LIN {X 0,Y 468.927,Z 382.309,A -85,B 0,C 180,E1 -7507.408,E2 -7507.408} C_VEL
LIN {X 0,Y 468.498,Z 392.429,A -85,B 0,C 180,E1 -7508.36,E2 -7508.36} C_VEL
LIN {X 0,Y 467.994,Z 402.327,A -85,B 0,C 180,E1 -7509.516,E2 -7509.516} C_VEL
LIN {X 0,Y 467.657,Z 410.813,A -85,B 0,C 180,E1 -7510.745,E2 -7510.745} C_VEL
LIN {X 0,Y 467.29,Z 417.675,A -85,B 0,C 180,E1 -7511.964,E2 -7511.964} C_VEL
LIN {X 0,Y 467.055,Z 424.349,A -85,B 0,C 180,E1 -7513.461,E2 -7513.461} C_VEL
LIN {X 0,Y 466.861,Z 429.589,A -85,B 0,C 180,E1 -7515.028,E2 -7515.028} C_VEL
LIN {X 0,Y 466.754,Z 432.659,A -85,B 0,C 180,E1 -7516.275,E2 -7516.275} C_VEL
LIN {X 0,Y 466.652,Z 434.866,A -85,B 0,C 180,E1 -7517.551,E2 -7517.551} C_VEL
LIN {X 0,Y 466.622,Z 436.188,A -85,B 0,C 180,E1 -7518.85,E2 -7518.85} C_VEL
LIN {X 0,Y 466.563,Z 436.605,A -85,B 0,C 180,E1 -7520.188,E2 -7520.188} C_VEL
LIN {X 0,Y 466.583,Z 435.757,A -85,B 0,C 180,E1 -7521.861,E2 -7521.861} C_VEL
LIN {X 0,Y 466.695,Z 433.486,A -85,B 0,C 180,E1 -7523.5,E2 -7523.5} C_VEL
LIN {X 0,Y 466.834,Z 429.723,A -85,B 0,C 180,E1 -7525.105,E2 -7525.105} C_VEL
LIN {X 0,Y 467.067,Z 424.472,A -85,B 0,C 180,E1 -7526.687,E2 -7526.687} C_VEL
LIN {X 0,Y 467.35,Z 418.59,A -85,B 0,C 180,E1 -7528.031,E2 -7528.031} C_VEL
LIN {X 0,Y 467.652,Z 411.787,A -85,B 0,C 180,E1 -7529.272,E2 -7529.272} C_VEL
LIN {X 0,Y 468.106,Z 402.57,A -85,B 0,C 180,E1 -7530.624,E2 -7530.624} C_VEL
LIN {X 0,Y 468.57,Z 393.367,A -85,B 0,C 180,E1 -7531.711,E2 -7531.711} C_VEL
LIN {X 0,Y 468.993,Z 383.202,A -85,B 0,C 180,E1 -7532.683,E2 -7532.683} C_VEL
LIN {X 0,Y 469.521,Z 371.519,A -85,B 0,C 180,E1 -7533.572,E2 -7533.572} C_VEL
LIN {X 0,Y 469.906,Z 360.613,A -85,B 0,C 180,E1 -7534.224,E2 -7534.224} C_VEL
LIN {X 0,Y 470.276,Z 347.828,A -85,B 0,C 180,E1 -7534.792,E2 -7534.792} C_VEL
LIN {X 0,Y 470.547,Z 334.524,A -85,B 0,C 180,E1 -7535.191,E2 -7535.191} C_VEL
LIN {X 0,Y 471.448,Z 240.188,A -85,B 0,C 180,E1 -7536.74,E2 -7536.74} C_VEL
LIN {X 0,Y 468.543,Z 226.096,A -85,B 0,C 180,E1 -7537.105,E2 -7537.105} C_VEL
LIN {X 0,Y 468.569,Z 216.391,A -85,B 0,C 180,E1 -7538.902,E2 -7538.902} C_VEL
LIN {X 0,Y 467.611,Z 211.239,A -85,B 0,C 180,E1 -7539.949,E2 -7539.949} C_VEL
LIN {X 0,Y 467.572,Z 211.241,A -85,B 0,C 180,E1 -7542.506,E2 -7542.506} C_VEL
LIN {X 0,Y 467.561,Z 211.248,A -85,B 0,C 180,E1 -7545.195,E2 -7545.195} C_VEL
LIN {X 0,Y 467.648,Z 211.236,A -85,B 0,C 180,E1 -7547.855,E2 -7547.855} C_VEL
LIN {X 0,Y 467.633,Z 211.238,A -85,B 0,C 180,E1 -7551.357,E2 -7551.357} C_VEL
LIN {X 0,Y 467.71,Z 211.223,A -85,B 0,C 180,E1 -7553.962,E2 -7553.962} C_VEL
LIN {X 0,Y 467.808,Z 211.214,A -85,B 0,C 180,E1 -7557.417,E2 -7557.417} C_VEL
LIN {X 0,Y 467.826,Z 211.208,A -85,B 0,C 180,E1 -7560,E2 -7560} C_VEL
LIN {X 0,Y 467.806,Z 211.213,A -85,B 0,C 180,E1 -7562.583,E2 -7562.583} C_VEL
LIN {X 0,Y 467.681,Z 211.223,A -85,B 0,C 180,E1 -7566.038,E2 -7566.038} C_VEL
LIN {X 0,Y 467.632,Z 211.235,A -85,B 0,C 180,E1 -7568.644,E2 -7568.644} C_VEL
LIN {X 0,Y 467.634,Z 211.23,A -85,B 0,C 180,E1 -7572.146,E2 -7572.146} C_VEL
LIN {X 0,Y 467.619,Z 211.233,A -85,B 0,C 180,E1 -7575.894,E2 -7575.894} C_VEL
LIN {X 0,Y 467.578,Z 211.238,A -85,B 0,C 180,E1 -7579.31,E2 -7579.31} C_VEL
LIN {X 0,Y 467.497,Z 211.25,A -85,B 0,C 180,E1 -7582.076,E2 -7582.076} C_VEL
LIN {X 0,Y 467.563,Z 211.244,A -85,B 0,C 180,E1 -7584.89,E2 -7584.89} C_VEL
LIN {X 0,Y 467.58,Z 211.237,A -85,B 0,C 180,E1 -7587.772,E2 -7587.772} C_VEL
LIN {X 0,Y 467.53,Z 211.245,A -85,B 0,C 180,E1 -7591.048,E2 -7591.048} C_VEL
LIN {X 0,Y 467.555,Z 211.246,A -85,B 0,C 180,E1 -7594.245,E2 -7594.245} C_VEL
LIN {X 0,Y 467.517,Z 211.246,A -85,B 0,C 180,E1 -7597.189,E2 -7597.189} C_VEL
LIN {X 0,Y 467.545,Z 211.247,A -85,B 0,C 180,E1 -7600.268,E2 -7600.268} C_VEL
LIN {X 0,Y 467.561,Z 211.242,A -85,B 0,C 180,E1 -7602.57,E2 -7602.57} C_VEL
LIN {X 0,Y 467.541,Z 211.242,A -85,B 0,C 180,E1 -7605.056,E2 -7605.056} C_VEL
LIN {X 0,Y 467.568,Z 211.24,A -85,B 0,C 180,E1 -7607.443,E2 -7607.443} C_VEL
LIN {X 0,Y 467.563,Z 211.241,A -85,B 0,C 180,E1 -7610.858,E2 -7610.858} C_VEL
LIN {X 0,Y 467.547,Z 211.247,A -85,B 0,C 180,E1 -7614.264,E2 -7614.264} C_VEL
LIN {X 0,Y 467.569,Z 211.242,A -85,B 0,C 180,E1 -7617.324,E2 -7617.324} C_VEL
LIN {X 0,Y 467.559,Z 211.245,A -85,B 0,C 180,E1 -7620.671,E2 -7620.671} C_VEL
LIN {X 0,Y 467.649,Z 211.353,A -85,B 0,C 180,E1 -7623.806,E2 -7623.806} C_VEL
LIN {X 0,Y 469.751,Z 222.852,A -85,B 0,C 180,E1 -7625.872,E2 -7625.872} C_VEL
LIN {X 0,Y 469.241,Z 237.693,A -85,B 0,C 180,E1 -7628.337,E2 -7628.337} C_VEL
LIN {X 0,Y 468.466,Z 259.202,A -85,B 0,C 180,E1 -7631.865,E2 -7631.865} C_VEL
LIN {X 0,Y 468.239,Z 265.745,A -85,B 0,C 180,E1 -7632.93,E2 -7632.93} C_VEL
LIN {X 0,Y 471.203,Z 287.173,A -85,B 0,C 180,E1 -7633.401,E2 -7633.401} C_VEL
LIN {X 0,Y 470.387,Z 375.627,A -85,B 0,C 180,E1 -7634.845,E2 -7634.845} C_VEL
LIN {X 0,Y 470.003,Z 387.734,A -85,B 0,C 180,E1 -7635.192,E2 -7635.192} C_VEL
LIN {X 0,Y 469.51,Z 401.066,A -85,B 0,C 180,E1 -7635.758,E2 -7635.758} C_VEL
LIN {X 0,Y 469.007,Z 413.098,A -85,B 0,C 180,E1 -7636.461,E2 -7636.461} C_VEL
LIN {X 0,Y 468.591,Z 424.153,A -85,B 0,C 180,E1 -7637.289,E2 -7637.289} C_VEL
LIN {X 0,Y 468.088,Z 435.073,A -85,B 0,C 180,E1 -7638.307,E2 -7638.307} C_VEL
LIN {X 0,Y 467.598,Z 444.443,A -85,B 0,C 180,E1 -7639.391,E2 -7639.391} C_VEL
LIN {X 0,Y 467.237,Z 453.554,A -85,B 0,C 180,E1 -7640.696,E2 -7640.696} C_VEL
LIN {X 0,Y 466.979,Z 460.9,A -85,B 0,C 180,E1 -7641.999,E2 -7641.999} C_VEL
LIN {X 0,Y 466.828,Z 465.861,A -85,B 0,C 180,E1 -7643.083,E2 -7643.083} C_VEL
LIN {X 0,Y 466.727,Z 470.686,A -85,B 0,C 180,E1 -7644.384,E2 -7644.384} C_VEL
LIN {X 0,Y 466.657,Z 474.379,A -85,B 0,C 180,E1 -7645.682,E2 -7645.682} C_VEL
LIN {X 0,Y 466.697,Z 476.289,A -85,B 0,C 180,E1 -7646.547,E2 -7646.547} C_VEL
LIN {X 0,Y 466.681,Z 477.722,A -85,B 0,C 180,E1 -7647.411,E2 -7647.411} C_VEL
LIN {X 0,Y 466.661,Z 478.748,A -85,B 0,C 180,E1 -7648.274,E2 -7648.274} C_VEL
LIN {X 0,Y 466.624,Z 479.377,A -85,B 0,C 180,E1 -7649.137,E2 -7649.137} C_VEL
LIN {X 0,Y 466.607,Z 479.604,A -85,B 0,C 180,E1 -7650,E2 -7650} C_VEL
LIN {X 0,Y 466.624,Z 479.391,A -85,B 0,C 180,E1 -7650.863,E2 -7650.863} C_VEL
LIN {X 0,Y 466.661,Z 478.783,A -85,B 0,C 180,E1 -7651.726,E2 -7651.726} C_VEL
LIN {X 0,Y 466.68,Z 477.779,A -85,B 0,C 180,E1 -7652.589,E2 -7652.589} C_VEL
LIN {X 0,Y 466.691,Z 476.357,A -85,B 0,C 180,E1 -7653.453,E2 -7653.453} C_VEL
LIN {X 0,Y 466.688,Z 473.375,A -85,B 0,C 180,E1 -7654.75,E2 -7654.75} C_VEL
LIN {X 0,Y 466.743,Z 469.333,A -85,B 0,C 180,E1 -7656.05,E2 -7656.05} C_VEL
LIN {X 0,Y 466.906,Z 463.103,A -85,B 0,C 180,E1 -7657.567,E2 -7657.567} C_VEL
LIN {X 0,Y 467.132,Z 456.305,A -85,B 0,C 180,E1 -7658.87,E2 -7658.87} C_VEL
LIN {X 0,Y 467.435,Z 447.857,A -85,B 0,C 180,E1 -7660.174,E2 -7660.174} C_VEL
LIN {X 0,Y 467.869,Z 439.152,A -85,B 0,C 180,E1 -7661.26,E2 -7661.26} C_VEL
LIN {X 0,Y 468.308,Z 428.98,A -85,B 0,C 180,E1 -7662.295,E2 -7662.295} C_VEL
LIN {X 0,Y 468.853,Z 417.789,A -85,B 0,C 180,E1 -7663.213,E2 -7663.213} C_VEL
LIN {X 0,Y 469.3,Z 405.934,A -85,B 0,C 180,E1 -7663.972,E2 -7663.972} C_VEL
LIN {X 0,Y 469.775,Z 393.641,A -85,B 0,C 180,E1 -7664.566,E2 -7664.566} C_VEL
LIN {X 0,Y 470.19,Z 380.174,A -85,B 0,C 180,E1 -7665.023,E2 -7665.023} C_VEL
LIN {X 0,Y 470.485,Z 365.01,A -85,B 0,C 180,E1 -7665.318,E2 -7665.318} C_VEL
LIN {X 0,Y 471.003,Z 285.344,A -85,B 0,C 180,E1 -7666.59,E2 -7666.59} C_VEL
LIN {X 0,Y 468.3,Z 266.657,A -85,B 0,C 180,E1 -7667.015,E2 -7667.015} C_VEL
LIN {X 0,Y 468.98,Z 247.902,A -85,B 0,C 180,E1 -7670.159,E2 -7670.159} C_VEL
LIN {X 0,Y 469.761,Z 230.47,A -85,B 0,C 180,E1 -7673.121,E2 -7673.121} C_VEL
LIN {X 0,Y 470.065,Z 224.101,A -85,B 0,C 180,E1 -7674.213,E2 -7674.213} C_VEL
LIN {X 0,Y 467.962,Z 212.85,A -85,B 0,C 180,E1 -7676.294,E2 -7676.294} C_VEL
LIN {X 0,Y 467.646,Z 211.235,A -85,B 0,C 180,E1 -7676.614,E2 -7676.614} C_VEL
LIN {X 0,Y 467.542,Z 211.247,A -85,B 0,C 180,E1 -7679.735,E2 -7679.735} C_VEL
LIN {X 0,Y 467.57,Z 211.238,A -85,B 0,C 180,E1 -7682.755,E2 -7682.755} C_VEL
LIN {X 0,Y 467.539,Z 211.249,A -85,B 0,C 180,E1 -7685.886,E2 -7685.886} C_VEL
LIN {X 0,Y 467.562,Z 211.239,A -85,B 0,C 180,E1 -7689.141,E2 -7689.141} C_VEL
LIN {X 0,Y 467.564,Z 211.239,A -85,B 0,C 180,E1 -7692.564,E2 -7692.564} C_VEL
LIN {X 0,Y 467.544,Z 211.242,A -85,B 0,C 180,E1 -7695.049,E2 -7695.049} C_VEL
LIN {X 0,Y 467.562,Z 211.243,A -85,B 0,C 180,E1 -7697.436,E2 -7697.436} C_VEL
LIN {X 0,Y 467.528,Z 211.243,A -85,B 0,C 180,E1 -7700.85,E2 -7700.85} C_VEL
LIN {X 0,Y 467.529,Z 211.244,A -85,B 0,C 180,E1 -7704.257,E2 -7704.257} C_VEL
LIN {X 0,Y 467.546,Z 211.246,A -85,B 0,C 180,E1 -7707.318,E2 -7707.318} C_VEL
LIN {X 0,Y 467.529,Z 211.243,A -85,B 0,C 180,E1 -7710.665,E2 -7710.665} C_VEL
LIN {X 0,Y 467.575,Z 211.242,A -85,B 0,C 180,E1 -7713.197,E2 -7713.197} C_VEL
LIN {X 0,Y 467.55,Z 211.24,A -85,B 0,C 180,E1 -7716.466,E2 -7716.466} C_VEL
LIN {X 0,Y 467.576,Z 211.24,A -85,B 0,C 180,E1 -7719.775,E2 -7719.775} C_VEL
LIN {X 0,Y 467.564,Z 211.239,A -85,B 0,C 180,E1 -7722.505,E2 -7722.505} C_VEL
LIN {X 0,Y 467.555,Z 211.248,A -85,B 0,C 180,E1 -7725.194,E2 -7725.194} C_VEL
LIN {X 0,Y 467.632,Z 211.231,A -85,B 0,C 180,E1 -7727.854,E2 -7727.854} C_VEL
LIN {X 0,Y 467.631,Z 211.235,A -85,B 0,C 180,E1 -7731.356,E2 -7731.356} C_VEL
LIN {X 0,Y 467.681,Z 211.224,A -85,B 0,C 180,E1 -7733.961,E2 -7733.961} C_VEL
LIN {X 0,Y 467.805,Z 211.211,A -85,B 0,C 180,E1 -7737.416,E2 -7737.416} C_VEL
LIN {X 0,Y 467.825,Z 211.206,A -85,B 0,C 180,E1 -7740,E2 -7740} C_VEL
LIN {X 0,Y 467.807,Z 211.213,A -85,B 0,C 180,E1 -7742.583,E2 -7742.583} C_VEL
LIN {X 0,Y 467.709,Z 211.221,A -85,B 0,C 180,E1 -7746.038,E2 -7746.038} C_VEL
LIN {X 0,Y 467.632,Z 211.237,A -85,B 0,C 180,E1 -7748.643,E2 -7748.643} C_VEL
LIN {X 0,Y 467.647,Z 211.23,A -85,B 0,C 180,E1 -7752.145,E2 -7752.145} C_VEL
LIN {X 0,Y 467.617,Z 211.233,A -85,B 0,C 180,E1 -7755.894,E2 -7755.894} C_VEL
LIN {X 0,Y 467.581,Z 211.237,A -85,B 0,C 180,E1 -7759.309,E2 -7759.309} C_VEL
LIN {X 0,Y 467.575,Z 211.24,A -85,B 0,C 180,E1 -7762.071,E2 -7762.071} C_VEL
LIN {X 0,Y 467.572,Z 211.24,A -85,B 0,C 180,E1 -7764.889,E2 -7764.889} C_VEL
LIN {X 0,Y 467.586,Z 211.237,A -85,B 0,C 180,E1 -7767.771,E2 -7767.771} C_VEL
LIN {X 0,Y 467.531,Z 211.243,A -85,B 0,C 180,E1 -7771.048,E2 -7771.048} C_VEL
LIN {X 0,Y 467.552,Z 211.248,A -85,B 0,C 180,E1 -7774.245,E2 -7774.245} C_VEL
LIN {X 0,Y 467.515,Z 211.245,A -85,B 0,C 180,E1 -7777.19,E2 -7777.19} C_VEL
LIN {X 0,Y 467.57,Z 211.245,A -85,B 0,C 180,E1 -7780.265,E2 -7780.265} C_VEL
LIN {X 0,Y 467.589,Z 211.238,A -85,B 0,C 180,E1 -7782.574,E2 -7782.574} C_VEL
LIN {X 0,Y 467.541,Z 211.241,A -85,B 0,C 180,E1 -7785.056,E2 -7785.056} C_VEL
LIN {X 0,Y 467.563,Z 211.24,A -85,B 0,C 180,E1 -7787.443,E2 -7787.443} C_VEL
LIN {X 0,Y 467.577,Z 211.237,A -85,B 0,C 180,E1 -7790.86,E2 -7790.86} C_VEL
LIN {X 0,Y 467.543,Z 211.245,A -85,B 0,C 180,E1 -7794.263,E2 -7794.263} C_VEL
LIN {X 0,Y 467.565,Z 211.24,A -85,B 0,C 180,E1 -7797.324,E2 -7797.324} C_VEL
LIN {X 0,Y 467.562,Z 211.239,A -85,B 0,C 180,E1 -7800.669,E2 -7800.669} C_VEL
LIN {X 0,Y 467.615,Z 211.234,A -85,B 0,C 180,E1 -7803.203,E2 -7803.203} C_VEL
LIN {X 0,Y 467.583,Z 211.236,A -85,B 0,C 180,E1 -7806.47,E2 -7806.47} C_VEL
LIN {X 0,Y 467.614,Z 211.238,A -85,B 0,C 180,E1 -7809.779,E2 -7809.779} C_VEL
LIN {X 0,Y 467.602,Z 211.234,A -85,B 0,C 180,E1 -7812.509,E2 -7812.509} C_VEL
LIN {X 0,Y 467.604,Z 211.238,A -85,B 0,C 180,E1 -7815.198,E2 -7815.198} C_VEL
LIN {X 0,Y 467.594,Z 211.237,A -85,B 0,C 180,E1 -7815.47,E2 -7815.47} C_VEL
LIN {X 0,Y 466.926,Z 211.32,A -85,B 0,C 180,E1 -7816.189,E2 -7816.189} C_VEL
LIN {X 0,Y 464.08,Z 211.68,A -85,B 0,C 180,E1 -7817.357,E2 -7817.357} C_VEL
LIN {X 0,Y 461.679,Z 211.974,A -85,B 0,C 180,E1 -7818.299,E2 -7818.299} C_VEL
LIN {X 0,Y 460.654,Z 212.102,A -85,B 0,C 180,E1 -7819.027,E2 -7819.027} C_VEL
LIN {X 0,Y 460.574,Z 212.114,A -85,B 0,C 180,E1 -7819.273,E2 -7819.273} C_VEL
LIN {X 0,Y 460.713,Z 212.092,A -85,B 0,C 180,E1 -7822.544,E2 -7822.544} C_VEL
LIN {X 0,Y 460.693,Z 212.096,A -85,B 0,C 180,E1 -7824.749,E2 -7824.749} C_VEL
LIN {X 0,Y 460.823,Z 212.085,A -85,B 0,C 180,E1 -7827.378,E2 -7827.378} C_VEL
LIN {X 0,Y 460.851,Z 212.075,A -85,B 0,C 180,E1 -7830,E2 -7830} C_VEL
LIN {X 0,Y 460.823,Z 212.08,A -85,B 0,C 180,E1 -7832.622,E2 -7832.622} C_VEL
LIN {X 0,Y 460.692,Z 212.095,A -85,B 0,C 180,E1 -7836.13,E2 -7836.13} C_VEL
LIN {X 0,Y 460.626,Z 212.107,A -85,B 0,C 180,E1 -7838.775,E2 -7838.775} C_VEL
LIN {X 0,Y 460.61,Z 212.107,A -85,B 0,C 180,E1 -7842.444,E2 -7842.444} C_VEL
LIN {X 0,Y 460.595,Z 212.107,A -85,B 0,C 180,E1 -7845.996,E2 -7845.996} C_VEL
LIN {X 0,Y 460.565,Z 212.118,A -85,B 0,C 180,E1 -7848.9,E2 -7848.9} C_VEL
LIN {X 0,Y 460.508,Z 212.118,A -85,B 0,C 180,E1 -7851.484,E2 -7851.484} C_VEL
LIN {X 0,Y 460.533,Z 212.117,A -85,B 0,C 180,E1 -7854.33,E2 -7854.33} C_VEL
LIN {X 0,Y 460.572,Z 212.114,A -85,B 0,C 180,E1 -7857.241,E2 -7857.241} C_VEL
LIN {X 0,Y 460.625,Z 212.228,A -85,B 0,C 180,E1 -7859.808,E2 -7859.808} C_VEL
LIN {X 0,Y 461.644,Z 218.347,A -85,B 0,C 180,E1 -7861.168,E2 -7861.168} C_VEL
LIN {X 0,Y 461.512,Z 226.254,A -85,B 0,C 180,E1 -7862.829,E2 -7862.829} C_VEL
LIN {X 0,Y 464.399,Z 240.609,A -85,B 0,C 180,E1 -7863.185,E2 -7863.185} C_VEL
LIN {X 0,Y 463.53,Z 333.526,A -85,B 0,C 180,E1 -7864.712,E2 -7864.712} C_VEL
LIN {X 0,Y 463.213,Z 346.696,A -85,B 0,C 180,E1 -7865.101,E2 -7865.101} C_VEL
LIN {X 0,Y 462.969,Z 358.713,A -85,B 0,C 180,E1 -7865.625,E2 -7865.625} C_VEL
LIN {X 0,Y 462.513,Z 370.891,A -85,B 0,C 180,E1 -7866.338,E2 -7866.338} C_VEL
LIN {X 0,Y 461.998,Z 382.253,A -85,B 0,C 180,E1 -7867.201,E2 -7867.201} C_VEL
LIN {X 0,Y 461.495,Z 393.331,A -85,B 0,C 180,E1 -7868.259,E2 -7868.259} C_VEL
LIN {X 0,Y 460.996,Z 402.697,A -85,B 0,C 180,E1 -7869.377,E2 -7869.377} C_VEL
LIN {X 0,Y 460.658,Z 411.115,A -85,B 0,C 180,E1 -7870.615,E2 -7870.615} C_VEL
LIN {X 0,Y 460.251,Z 418.028,A -85,B 0,C 180,E1 -7871.861,E2 -7871.861} C_VEL
LIN {X 0,Y 460.052,Z 423.596,A -85,B 0,C 180,E1 -7873.102,E2 -7873.102} C_VEL
LIN {X 0,Y 459.825,Z 429.07,A -85,B 0,C 180,E1 -7874.667,E2 -7874.667} C_VEL
LIN {X 0,Y 459.711,Z 432.36,A -85,B 0,C 180,E1 -7875.927,E2 -7875.927} C_VEL
LIN {X 0,Y 459.55,Z 435.433,A -85,B 0,C 180,E1 -7877.709,E2 -7877.709} C_VEL
LIN {X 0,Y 459.527,Z 436.537,A -85,B 0,C 180,E1 -7878.88,E2 -7878.88} C_VEL
LIN {X 0,Y 459.489,Z 436.946,A -85,B 0,C 180,E1 -7880.029,E2 -7880.029} C_VEL
LIN {X 0,Y 459.478,Z 436.581,A -85,B 0,C 180,E1 -7881.26,E2 -7881.26} C_VEL
LIN {X 0,Y 459.514,Z 435.203,A -85,B 0,C 180,E1 -7882.676,E2 -7882.676} C_VEL
LIN {X 0,Y 459.678,Z 432.697,A -85,B 0,C 180,E1 -7884.118,E2 -7884.118} C_VEL
LIN {X 0,Y 459.807,Z 428.84,A -85,B 0,C 180,E1 -7885.617,E2 -7885.617} C_VEL
LIN {X 0,Y 460.092,Z 423.407,A -85,B 0,C 180,E1 -7887.145,E2 -7887.145} C_VEL
LIN {X 0,Y 460.399,Z 417.313,A -85,B 0,C 180,E1 -7888.479,E2 -7888.479} C_VEL
LIN {X 0,Y 460.784,Z 409.913,A -85,B 0,C 180,E1 -7889.78,E2 -7889.78} C_VEL
LIN {X 0,Y 461.267,Z 400.737,A -85,B 0,C 180,E1 -7891.07,E2 -7891.07} C_VEL
LIN {X 0,Y 461.727,Z 390.638,A -85,B 0,C 180,E1 -7892.213,E2 -7892.213} C_VEL
LIN {X 0,Y 462.284,Z 379.757,A -85,B 0,C 180,E1 -7893.198,E2 -7893.198} C_VEL
LIN {X 0,Y 462.807,Z 367.681,A -85,B 0,C 180,E1 -7894.054,E2 -7894.054} C_VEL
LIN {X 0,Y 463.221,Z 356.195,A -85,B 0,C 180,E1 -7894.681,E2 -7894.681} C_VEL
LIN {X 0,Y 463.538,Z 343.535,A -85,B 0,C 180,E1 -7895.186,E2 -7895.186} C_VEL
LIN {X 0,Y 463.781,Z 329.939,A -85,B 0,C 180,E1 -7895.529,E2 -7895.529} C_VEL
LIN {X 0,Y 464.699,Z 241.15,A -85,B 0,C 180,E1 -7896.993,E2 -7896.993} C_VEL
LIN {X 0,Y 461.648,Z 226.372,A -85,B 0,C 180,E1 -7897.394,E2 -7897.394} C_VEL
LIN {X 0,Y 461.632,Z 217.605,A -85,B 0,C 180,E1 -7899.037,E2 -7899.037} C_VEL
LIN {X 0,Y 460.568,Z 212.116,A -85,B 0,C 180,E1 -7900.153,E2 -7900.153} C_VEL
LIN {X 0,Y 460.527,Z 212.123,A -85,B 0,C 180,E1 -7903.145,E2 -7903.145} C_VEL
LIN {X 0,Y 460.515,Z 212.125,A -85,B 0,C 180,E1 -7905.867,E2 -7905.867} C_VEL
LIN {X 0,Y 460.589,Z 212.114,A -85,B 0,C 180,E1 -7908.559,E2 -7908.559} C_VEL
LIN {X 0,Y 460.647,Z 212.103,A -85,B 0,C 180,E1 -7912.108,E2 -7912.108} C_VEL
LIN {X 0,Y 460.656,Z 212.104,A -85,B 0,C 180,E1 -7914.748,E2 -7914.748} C_VEL
LIN {X 0,Y 460.749,Z 212.094,A -85,B 0,C 180,E1 -7917.378,E2 -7917.378} C_VEL
LIN {X 0,Y 460.797,Z 212.084,A -85,B 0,C 180,E1 -7920,E2 -7920} C_VEL
LIN {X 0,Y 460.748,Z 212.093,A -85,B 0,C 180,E1 -7922.623,E2 -7922.623} C_VEL
LIN {X 0,Y 460.648,Z 212.099,A -85,B 0,C 180,E1 -7926.131,E2 -7926.131} C_VEL
LIN {X 0,Y 460.58,Z 212.113,A -85,B 0,C 180,E1 -7928.777,E2 -7928.777} C_VEL
LIN {X 0,Y 460.588,Z 212.11,A -85,B 0,C 180,E1 -7932.458,E2 -7932.458} C_VEL
LIN {X 0,Y 460.577,Z 212.11,A -85,B 0,C 180,E1 -7936.009,E2 -7936.009} C_VEL
LIN {X 0,Y 460.524,Z 212.116,A -85,B 0,C 180,E1 -7939.618,E2 -7939.618} C_VEL
LIN {X 0,Y 460.472,Z 212.129,A -85,B 0,C 180,E1 -7942.431,E2 -7942.431} C_VEL
LIN {X 0,Y 460.527,Z 212.117,A -85,B 0,C 180,E1 -7945.804,E2 -7945.804} C_VEL
LIN {X 0,Y 460.513,Z 212.121,A -85,B 0,C 180,E1 -7948.236,E2 -7948.236} C_VEL
LIN {X 0,Y 460.484,Z 212.122,A -85,B 0,C 180,E1 -7951.286,E2 -7951.286} C_VEL
LIN {X 0,Y 460.5,Z 212.124,A -85,B 0,C 180,E1 -7954.509,E2 -7954.509} C_VEL
LIN {X 0,Y 460.47,Z 212.124,A -85,B 0,C 180,E1 -7957.626,E2 -7957.626} C_VEL
LIN {X 0,Y 460.51,Z 212.123,A -85,B 0,C 180,E1 -7960.272,E2 -7960.272} C_VEL
LIN {X 0,Y 460.47,Z 212.122,A -85,B 0,C 180,E1 -7963.379,E2 -7963.379} C_VEL
LIN {X 0,Y 460.473,Z 212.125,A -85,B 0,C 180,E1 -7966.627,E2 -7966.627} C_VEL
LIN {X 0,Y 460.522,Z 212.12,A -85,B 0,C 180,E1 -7969.734,E2 -7969.734} C_VEL
LIN {X 0,Y 460.483,Z 212.125,A -85,B 0,C 180,E1 -7972.527,E2 -7972.527} C_VEL
LIN {X 0,Y 460.534,Z 212.119,A -85,B 0,C 180,E1 -7975.627,E2 -7975.627} C_VEL
LIN {X 0,Y 460.526,Z 212.119,A -85,B 0,C 180,E1 -7978.747,E2 -7978.747} C_VEL
LIN {X 0,Y 460.572,Z 212.118,A -85,B 0,C 180,E1 -7982.257,E2 -7982.257} C_VEL
LIN {X 0,Y 460.601,Z 212.258,A -85,B 0,C 180,E1 -7983.588,E2 -7983.588} C_VEL
LIN {X 0,Y 462.485,Z 221.848,A -85,B 0,C 180,E1 -7985.349,E2 -7985.349} C_VEL
LIN {X 0,Y 462.843,Z 225.754,A -85,B 0,C 180,E1 -7986.037,E2 -7986.037} C_VEL
LIN {X 0,Y 462.101,Z 242.367,A -85,B 0,C 180,E1 -7988.828,E2 -7988.828} C_VEL
LIN {X 0,Y 461.371,Z 263.03,A -85,B 0,C 180,E1 -7992.264,E2 -7992.264} C_VEL
LIN {X 0,Y 461.288,Z 265.345,A -85,B 0,C 180,E1 -7992.646,E2 -7992.646} C_VEL
LIN {X 0,Y 464.425,Z 287.456,A -85,B 0,C 180,E1 -7993.15,E2 -7993.15} C_VEL
LIN {X 0,Y 463.543,Z 375.457,A -85,B 0,C 180,E1 -7994.615,E2 -7994.615} C_VEL
LIN {X 0,Y 463.121,Z 388.241,A -85,B 0,C 180,E1 -7994.995,E2 -7994.995} C_VEL
LIN {X 0,Y 462.599,Z 400.776,A -85,B 0,C 180,E1 -7995.54,E2 -7995.54} C_VEL
LIN {X 0,Y 462.085,Z 412.792,A -85,B 0,C 180,E1 -7996.254,E2 -7996.254} C_VEL
LIN {X 0,Y 461.589,Z 424.834,A -85,B 0,C 180,E1 -7997.178,E2 -7997.178} C_VEL
LIN {X 0,Y 461.1,Z 434.754,A -85,B 0,C 180,E1 -7998.127,E2 -7998.127} C_VEL
LIN {X 0,Y 460.586,Z 444.117,A -85,B 0,C 180,E1 -7999.228,E2 -7999.228} C_VEL
LIN {X 0,Y 460.177,Z 453.224,A -85,B 0,C 180,E1 -8000.552,E2 -8000.552} C_VEL
LIN {X 0,Y 459.906,Z 460.57,A -85,B 0,C 180,E1 -8001.875,E2 -8001.875} C_VEL
LIN {X 0,Y 459.72,Z 466.815,A -85,B 0,C 180,E1 -8003.295,E2 -8003.295} C_VEL
LIN {X 0,Y 459.64,Z 471.707,A -85,B 0,C 180,E1 -8004.737,E2 -8004.737} C_VEL
LIN {X 0,Y 459.572,Z 474.055,A -85,B 0,C 180,E1 -8005.615,E2 -8005.615} C_VEL
LIN {X 0,Y 459.594,Z 475.965,A -85,B 0,C 180,E1 -8006.494,E2 -8006.494} C_VEL
LIN {X 0,Y 459.601,Z 477.398,A -85,B 0,C 180,E1 -8007.371,E2 -8007.371} C_VEL
LIN {X 0,Y 459.57,Z 478.423,A -85,B 0,C 180,E1 -8008.247,E2 -8008.247} C_VEL
LIN {X 0,Y 459.557,Z 479.053,A -85,B 0,C 180,E1 -8009.124,E2 -8009.124} C_VEL
LIN {X 0,Y 459.538,Z 479.277,A -85,B 0,C 180,E1 -8010,E2 -8010} C_VEL
LIN {X 0,Y 459.557,Z 479.061,A -85,B 0,C 180,E1 -8010.876,E2 -8010.876} C_VEL
LIN {X 0,Y 459.57,Z 478.45,A -85,B 0,C 180,E1 -8011.752,E2 -8011.752} C_VEL
LIN {X 0,Y 459.6,Z 477.443,A -85,B 0,C 180,E1 -8012.629,E2 -8012.629} C_VEL
LIN {X 0,Y 459.589,Z 476.013,A -85,B 0,C 180,E1 -8013.506,E2 -8013.506} C_VEL
LIN {X 0,Y 459.618,Z 473.025,A -85,B 0,C 180,E1 -8014.824,E2 -8014.824} C_VEL
LIN {X 0,Y 459.714,Z 467.911,A -85,B 0,C 180,E1 -8016.43,E2 -8016.43} C_VEL
LIN {X 0,Y 459.87,Z 461.699,A -85,B 0,C 180,E1 -8017.905,E2 -8017.905} C_VEL
LIN {X 0,Y 460.152,Z 454.642,A -85,B 0,C 180,E1 -8019.227,E2 -8019.227} C_VEL
LIN {X 0,Y 460.491,Z 445.789,A -85,B 0,C 180,E1 -8020.552,E2 -8020.552} C_VEL
LIN {X 0,Y 461.058,Z 435.745,A -85,B 0,C 180,E1 -8021.762,E2 -8021.762} C_VEL
LIN {X 0,Y 461.561,Z 424.877,A -85,B 0,C 180,E1 -8022.806,E2 -8022.806} C_VEL
LIN {X 0,Y 462.04,Z 414.123,A -85,B 0,C 180,E1 -8023.635,E2 -8023.635} C_VEL
LIN {X 0,Y 462.553,Z 402.351,A -85,B 0,C 180,E1 -8024.349,E2 -8024.349} C_VEL
LIN {X 0,Y 463.027,Z 389.502,A -85,B 0,C 180,E1 -8024.923,E2 -8024.923} C_VEL
LIN {X 0,Y 463.403,Z 375.882,A -85,B 0,C 180,E1 -8025.333,E2 -8025.333} C_VEL
LIN {X 0,Y 464.134,Z 301.407,A -85,B 0,C 180,E1 -8026.559,E2 -8026.559} C_VEL
LIN {X 0,Y 464.135,Z 286.017,A -85,B 0,C 180,E1 -8026.816,E2 -8026.816} C_VEL
LIN {X 0,Y 461.311,Z 266.427,A -85,B 0,C 180,E1 -8027.256,E2 -8027.256} C_VEL
LIN {X 0,Y 462.007,Z 248.892,A -85,B 0,C 180,E1 -8030.245,E2 -8030.245} C_VEL
LIN {X 0,Y 462.824,Z 231.449,A -85,B 0,C 180,E1 -8033.251,E2 -8033.251} C_VEL
LIN {X 0,Y 463.057,Z 224.843,A -85,B 0,C 180,E1 -8034.405,E2 -8034.405} C_VEL
LIN {X 0,Y 460.629,Z 212.109,A -85,B 0,C 180,E1 -8036.838,E2 -8036.838} C_VEL
LIN {X 0,Y 460.499,Z 212.126,A -85,B 0,C 180,E1 -8040.237,E2 -8040.237} C_VEL
LIN {X 0,Y 460.515,Z 212.117,A -85,B 0,C 180,E1 -8043.322,E2 -8043.322} C_VEL
LIN {X 0,Y 460.461,Z 212.125,A -85,B 0,C 180,E1 -8046.526,E2 -8046.526} C_VEL
LIN {X 0,Y 460.512,Z 212.125,A -85,B 0,C 180,E1 -8049.859,E2 -8049.859} C_VEL
LIN {X 0,Y 460.489,Z 212.12,A -85,B 0,C 180,E1 -8052.897,E2 -8052.897} C_VEL
LIN {X 0,Y 460.485,Z 212.128,A -85,B 0,C 180,E1 -8055.827,E2 -8055.827} C_VEL
LIN {X 0,Y 460.501,Z 212.119,A -85,B 0,C 180,E1 -8058.985,E2 -8058.985} C_VEL
LIN {X 0,Y 460.487,Z 212.123,A -85,B 0,C 180,E1 -8061.263,E2 -8061.263} C_VEL
LIN {X 0,Y 460.479,Z 212.121,A -85,B 0,C 180,E1 -8064.551,E2 -8064.551} C_VEL
LIN {X 0,Y 460.495,Z 212.125,A -85,B 0,C 180,E1 -8067.712,E2 -8067.712} C_VEL
LIN {X 0,Y 460.499,Z 212.119,A -85,B 0,C 180,E1 -8070.766,E2 -8070.766} C_VEL
LIN {X 0,Y 460.522,Z 212.12,A -85,B 0,C 180,E1 -8073.732,E2 -8073.732} C_VEL
LIN {X 0,Y 460.504,Z 212.119,A -85,B 0,C 180,E1 -8076.621,E2 -8076.621} C_VEL
LIN {X 0,Y 460.507,Z 212.124,A -85,B 0,C 180,E1 -8079.45,E2 -8079.45} C_VEL
LIN {X 0,Y 460.513,Z 212.117,A -85,B 0,C 180,E1 -8082.228,E2 -8082.228} C_VEL
LIN {X 0,Y 460.515,Z 212.121,A -85,B 0,C 180,E1 -8084.963,E2 -8084.963} C_VEL
LIN {X 0,Y 460.58,Z 212.111,A -85,B 0,C 180,E1 -8087.665,E2 -8087.665} C_VEL
LIN {X 0,Y 460.579,Z 212.115,A -85,B 0,C 180,E1 -8091.223,E2 -8091.223} C_VEL
LIN {X 0,Y 460.647,Z 212.1,A -85,B 0,C 180,E1 -8093.869,E2 -8093.869} C_VEL
LIN {X 0,Y 460.747,Z 212.091,A -85,B 0,C 180,E1 -8097.377,E2 -8097.377} C_VEL
LIN {X 0,Y 460.796,Z 212.082,A -85,B 0,C 180,E1 -8100,E2 -8100} C_VEL
LIN {X 0,Y 460.748,Z 212.092,A -85,B 0,C 180,E1 -8102.622,E2 -8102.622} C_VEL
LIN {X 0,Y 460.675,Z 212.098,A -85,B 0,C 180,E1 -8106.13,E2 -8106.13} C_VEL
LIN {X 0,Y 460.58,Z 212.117,A -85,B 0,C 180,E1 -8108.777,E2 -8108.777} C_VEL
LIN {X 0,Y 460.585,Z 212.113,A -85,B 0,C 180,E1 -8112.458,E2 -8112.458} C_VEL
LIN {X 0,Y 460.575,Z 212.111,A -85,B 0,C 180,E1 -8116.008,E2 -8116.008} C_VEL
LIN {X 0,Y 460.53,Z 212.115,A -85,B 0,C 180,E1 -8119.617,E2 -8119.617} C_VEL
LIN {X 0,Y 460.526,Z 212.122,A -85,B 0,C 180,E1 -8122.428,E2 -8122.428} C_VEL
LIN {X 0,Y 460.542,Z 212.114,A -85,B 0,C 180,E1 -8125.809,E2 -8125.809} C_VEL
LIN {X 0,Y 460.516,Z 212.123,A -85,B 0,C 180,E1 -8128.235,E2 -8128.235} C_VEL
LIN {X 0,Y 460.483,Z 212.121,A -85,B 0,C 180,E1 -8131.286,E2 -8131.286} C_VEL
LIN {X 0,Y 460.496,Z 212.124,A -85,B 0,C 180,E1 -8134.508,E2 -8134.508} C_VEL
LIN {X 0,Y 460.496,Z 212.12,A -85,B 0,C 180,E1 -8137.623,E2 -8137.623} C_VEL
LIN {X 0,Y 460.532,Z 212.121,A -85,B 0,C 180,E1 -8140.276,E2 -8140.276} C_VEL
LIN {X 0,Y 460.495,Z 212.12,A -85,B 0,C 180,E1 -8143.376,E2 -8143.376} C_VEL
LIN {X 0,Y 460.472,Z 212.123,A -85,B 0,C 180,E1 -8146.628,E2 -8146.628} C_VEL
LIN {X 0,Y 460.534,Z 212.119,A -85,B 0,C 180,E1 -8149.731,E2 -8149.731} C_VEL
LIN {X 0,Y 460.506,Z 212.119,A -85,B 0,C 180,E1 -8152.522,E2 -8152.522} C_VEL
LIN {X 0,Y 460.53,Z 212.12,A -85,B 0,C 180,E1 -8155.627,E2 -8155.627} C_VEL
LIN {X 0,Y 460.521,Z 212.116,A -85,B 0,C 180,E1 -8158.747,E2 -8158.747} C_VEL
LIN {X 0,Y 460.576,Z 212.111,A -85,B 0,C 180,E1 -8162.255,E2 -8162.255} C_VEL
LIN {X 0,Y 460.548,Z 212.113,A -85,B 0,C 180,E1 -8164.708,E2 -8164.708} C_VEL
LIN {X 0,Y 460.503,Z 212.126,A -85,B 0,C 180,E1 -8167.574,E2 -8167.574} C_VEL
LIN {X 0,Y 460.561,Z 212.111,A -85,B 0,C 180,E1 -8170.387,E2 -8170.387} C_VEL
LIN {X 0,Y 460.559,Z 212.114,A -85,B 0,C 180,E1 -8173.148,E2 -8173.148} C_VEL
LIN {X 0,Y 460.553,Z 212.115,A -85,B 0,C 180,E1 -8175.87,E2 -8175.87} C_VEL
LIN {X 0,Y 460.608,Z 212.105,A -85,B 0,C 180,E1 -8178.561,E2 -8178.561} C_VEL
LIN {X 0,Y 460.574,Z 212.114,A -85,B 0,C 180,E1 -8179.273,E2 -8179.273} C_VEL
LIN {X 0,Y 459.922,Z 212.202,A -85,B 0,C 180,E1 -8180.003,E2 -8180.003} C_VEL
LIN {X 0,Y 457.1,Z 212.554,A -85,B 0,C 180,E1 -8181.19,E2 -8181.19} C_VEL
LIN {X 0,Y 454.716,Z 212.845,A -85,B 0,C 180,E1 -8182.147,E2 -8182.147} C_VEL
LIN {X 0,Y 453.704,Z 212.968,A -85,B 0,C 180,E1 -8182.886,E2 -8182.886} C_VEL
LIN {X 0,Y 453.627,Z 212.976,A -85,B 0,C 180,E1 -8183.136,E2 -8183.136} C_VEL
LIN {X 0,Y 453.666,Z 212.971,A -85,B 0,C 180,E1 -8184.667,E2 -8184.667} C_VEL
LIN {X 0,Y 453.763,Z 212.965,A -85,B 0,C 180,E1 -8187.337,E2 -8187.337} C_VEL
LIN {X 0,Y 453.822,Z 212.951,A -85,B 0,C 180,E1 -8190,E2 -8190} C_VEL
LIN {X 0,Y 453.764,Z 212.96,A -85,B 0,C 180,E1 -8192.663,E2 -8192.663} C_VEL
LIN {X 0,Y 453.659,Z 212.971,A -85,B 0,C 180,E1 -8196.225,E2 -8196.225} C_VEL
LIN {X 0,Y 453.59,Z 212.986,A -85,B 0,C 180,E1 -8198.912,E2 -8198.912} C_VEL
LIN {X 0,Y 453.56,Z 212.986,A -85,B 0,C 180,E1 -8202.528,E2 -8202.528} C_VEL
LIN {X 0,Y 453.54,Z 212.986,A -85,B 0,C 180,E1 -8206.194,E2 -8206.194} C_VEL
LIN {X 0,Y 453.514,Z 212.994,A -85,B 0,C 180,E1 -8209.039,E2 -8209.039} C_VEL
LIN {X 0,Y 453.468,Z 212.995,A -85,B 0,C 180,E1 -8211.834,E2 -8211.834} C_VEL
LIN {X 0,Y 453.504,Z 212.998,A -85,B 0,C 180,E1 -8214.732,E2 -8214.732} C_VEL
LIN {X 0,Y 453.528,Z 212.991,A -85,B 0,C 180,E1 -8217.959,E2 -8217.959} C_VEL
LIN {X 0,Y 453.589,Z 213.176,A -85,B 0,C 180,E1 -8219.656,E2 -8219.656} C_VEL
LIN {X 0,Y 454.707,Z 219.963,A -85,B 0,C 180,E1 -8221.18,E2 -8221.18} C_VEL
LIN {X 0,Y 454.57,Z 226.527,A -85,B 0,C 180,E1 -8222.576,E2 -8222.576} C_VEL
LIN {X 0,Y 457.656,Z 242.228,A -85,B 0,C 180,E1 -8222.967,E2 -8222.967} C_VEL
LIN {X 0,Y 456.682,Z 333.247,A -85,B 0,C 180,E1 -8224.482,E2 -8224.482} C_VEL
LIN {X 0,Y 456.332,Z 346.852,A -85,B 0,C 180,E1 -8224.884,E2 -8224.884} C_VEL
LIN {X 0,Y 456.072,Z 358.931,A -85,B 0,C 180,E1 -8225.418,E2 -8225.418} C_VEL
LIN {X 0,Y 455.596,Z 371.096,A -85,B 0,C 180,E1 -8226.139,E2 -8226.139} C_VEL
LIN {X 0,Y 455.042,Z 382.699,A -85,B 0,C 180,E1 -8227.033,E2 -8227.033} C_VEL
LIN {X 0,Y 454.562,Z 393.181,A -85,B 0,C 180,E1 -8228.047,E2 -8228.047} C_VEL
LIN {X 0,Y 454.116,Z 401.562,A -85,B 0,C 180,E1 -8229.037,E2 -8229.037} C_VEL
LIN {X 0,Y 453.722,Z 410.216,A -85,B 0,C 180,E1 -8230.287,E2 -8230.287} C_VEL
LIN {X 0,Y 453.285,Z 417.133,A -85,B 0,C 180,E1 -8231.51,E2 -8231.51} C_VEL
LIN {X 0,Y 453.002,Z 424.05,A -85,B 0,C 180,E1 -8233.044,E2 -8233.044} C_VEL
LIN {X 0,Y 452.788,Z 428.925,A -85,B 0,C 180,E1 -8234.44,E2 -8234.44} C_VEL
LIN {X 0,Y 452.644,Z 432.219,A -85,B 0,C 180,E1 -8235.678,E2 -8235.678} C_VEL
LIN {X 0,Y 452.54,Z 434.618,A -85,B 0,C 180,E1 -8236.896,E2 -8236.896} C_VEL
LIN {X 0,Y 452.45,Z 436.327,A -85,B 0,C 180,E1 -8238.203,E2 -8238.203} C_VEL
LIN {X 0,Y 452.401,Z 437.179,A -85,B 0,C 180,E1 -8239.564,E2 -8239.564} C_VEL
LIN {X 0,Y 452.394,Z 437.083,A -85,B 0,C 180,E1 -8240.957,E2 -8240.957} C_VEL
LIN {X 0,Y 452.446,Z 435.551,A -85,B 0,C 180,E1 -8242.714,E2 -8242.714} C_VEL
LIN {X 0,Y 452.64,Z 432.586,A -85,B 0,C 180,E1 -8244.397,E2 -8244.397} C_VEL
LIN {X 0,Y 452.793,Z 428.17,A -85,B 0,C 180,E1 -8246.03,E2 -8246.03} C_VEL
LIN {X 0,Y 453.095,Z 423.252,A -85,B 0,C 180,E1 -8247.384,E2 -8247.384} C_VEL
LIN {X 0,Y 453.466,Z 416.373,A -85,B 0,C 180,E1 -8248.871,E2 -8248.871} C_VEL
LIN {X 0,Y 453.862,Z 409.104,A -85,B 0,C 180,E1 -8250.119,E2 -8250.119} C_VEL
LIN {X 0,Y 454.362,Z 400.294,A -85,B 0,C 180,E1 -8251.347,E2 -8251.347} C_VEL
LIN {X 0,Y 454.891,Z 389.992,A -85,B 0,C 180,E1 -8252.512,E2 -8252.512} C_VEL
LIN {X 0,Y 455.453,Z 379.022,A -85,B 0,C 180,E1 -8253.494,E2 -8253.494} C_VEL
LIN {X 0,Y 455.986,Z 367.482,A -85,B 0,C 180,E1 -8254.312,E2 -8254.312} C_VEL
LIN {X 0,Y 456.434,Z 355.794,A -85,B 0,C 180,E1 -8254.95,E2 -8254.95} C_VEL
LIN {X 0,Y 456.779,Z 342.928,A -85,B 0,C 180,E1 -8255.454,E2 -8255.454} C_VEL
LIN {X 0,Y 456.976,Z 330.626,A -85,B 0,C 180,E1 -8255.768,E2 -8255.768} C_VEL
LIN {X 0,Y 457.926,Z 241.904,A -85,B 0,C 180,E1 -8257.261,E2 -8257.261} C_VEL
LIN {X 0,Y 454.761,Z 226.729,A -85,B 0,C 180,E1 -8257.678,E2 -8257.678} C_VEL
LIN {X 0,Y 454.702,Z 218.863,A -85,B 0,C 180,E1 -8259.177,E2 -8259.177} C_VEL
LIN {X 0,Y 453.507,Z 212.996,A -85,B 0,C 180,E1 -8260.391,E2 -8260.391} C_VEL
LIN {X 0,Y 453.53,Z 212.994,A -85,B 0,C 180,E1 -8263.875,E2 -8263.875} C_VEL
LIN {X 0,Y 453.555,Z 212.994,A -85,B 0,C 180,E1 -8267.471,E2 -8267.471} C_VEL
LIN {X 0,Y 453.545,Z 212.994,A -85,B 0,C 180,E1 -8271.086,E2 -8271.086} C_VEL
LIN {X 0,Y 453.643,Z 212.977,A -85,B 0,C 180,E1 -8273.775,E2 -8273.775} C_VEL
LIN {X 0,Y 453.694,Z 212.974,A -85,B 0,C 180,E1 -8277.337,E2 -8277.337} C_VEL
LIN {X 0,Y 453.768,Z 212.959,A -85,B 0,C 180,E1 -8280,E2 -8280} C_VEL
LIN {X 0,Y 453.692,Z 212.972,A -85,B 0,C 180,E1 -8282.664,E2 -8282.664} C_VEL
LIN {X 0,Y 453.616,Z 212.976,A -85,B 0,C 180,E1 -8286.226,E2 -8286.226} C_VEL
LIN {X 0,Y 453.544,Z 212.99,A -85,B 0,C 180,E1 -8288.915,E2 -8288.915} C_VEL
LIN {X 0,Y 453.556,Z 212.987,A -85,B 0,C 180,E1 -8292.552,E2 -8292.552} C_VEL
LIN {X 0,Y 453.512,Z 212.992,A -85,B 0,C 180,E1 -8296.197,E2 -8296.197} C_VEL
LIN {X 0,Y 453.474,Z 212.998,A -85,B 0,C 180,E1 -8299.042,E2 -8299.042} C_VEL
LIN {X 0,Y 453.436,Z 213,A -85,B 0,C 180,E1 -8301.839,E2 -8301.839} C_VEL
LIN {X 0,Y 453.473,Z 213.001,A -85,B 0,C 180,E1 -8304.737,E2 -8304.737} C_VEL
LIN {X 0,Y 453.493,Z 212.993,A -85,B 0,C 180,E1 -8307.962,E2 -8307.962} C_VEL
LIN {X 0,Y 453.429,Z 213,A -85,B 0,C 180,E1 -8311.528,E2 -8311.528} C_VEL
LIN {X 0,Y 453.456,Z 212.998,A -85,B 0,C 180,E1 -8314.78,E2 -8314.78} C_VEL
LIN {X 0,Y 453.43,Z 213.004,A -85,B 0,C 180,E1 -8318.315,E2 -8318.315} C_VEL
LIN {X 0,Y 453.467,Z 212.999,A -85,B 0,C 180,E1 -8320.612,E2 -8320.612} C_VEL
LIN {X 0,Y 453.436,Z 213.006,A -85,B 0,C 180,E1 -8324.225,E2 -8324.225} C_VEL
LIN {X 0,Y 453.439,Z 212.999,A -85,B 0,C 180,E1 -8327.008,E2 -8327.008} C_VEL
LIN {X 0,Y 453.475,Z 212.996,A -85,B 0,C 180,E1 -8329.412,E2 -8329.412} C_VEL
LIN {X 0,Y 453.433,Z 213.007,A -85,B 0,C 180,E1 -8332.231,E2 -8332.231} C_VEL
LIN {X 0,Y 453.474,Z 212.995,A -85,B 0,C 180,E1 -8335.226,E2 -8335.226} C_VEL
LIN {X 0,Y 453.454,Z 213.002,A -85,B 0,C 180,E1 -8338.478,E2 -8338.478} C_VEL
LIN {X 0,Y 453.523,Z 212.996,A -85,B 0,C 180,E1 -8342.043,E2 -8342.043} C_VEL
LIN {X 0,Y 453.583,Z 213.107,A -85,B 0,C 180,E1 -8343.348,E2 -8343.348} C_VEL
LIN {X 0,Y 455.677,Z 224.068,A -85,B 0,C 180,E1 -8345.394,E2 -8345.394} C_VEL
LIN {X 0,Y 455.85,Z 228.277,A -85,B 0,C 180,E1 -8346.135,E2 -8346.135} C_VEL
LIN {X 0,Y 455.06,Z 244.876,A -85,B 0,C 180,E1 -8348.959,E2 -8348.959} C_VEL
LIN {X 0,Y 454.342,Z 264.934,A -85,B 0,C 180,E1 -8352.346,E2 -8352.346} C_VEL
LIN {X 0,Y 457.66,Z 288.102,A -85,B 0,C 180,E1 -8352.894,E2 -8352.894} C_VEL
LIN {X 0,Y 456.743,Z 374.285,A -85,B 0,C 180,E1 -8354.352,E2 -8354.352} C_VEL
LIN {X 0,Y 456.296,Z 387.323,A -85,B 0,C 180,E1 -8354.737,E2 -8354.737} C_VEL
LIN {X 0,Y 455.727,Z 400.554,A -85,B 0,C 180,E1 -8355.317,E2 -8355.317} C_VEL
LIN {X 0,Y 455.179,Z 412.525,A -85,B 0,C 180,E1 -8356.041,E2 -8356.041} C_VEL
LIN {X 0,Y 454.632,Z 424.544,A -85,B 0,C 180,E1 -8356.979,E2 -8356.979} C_VEL
LIN {X 0,Y 454.109,Z 434.449,A -85,B 0,C 180,E1 -8357.942,E2 -8357.942} C_VEL
LIN {X 0,Y 453.588,Z 443.802,A -85,B 0,C 180,E1 -8359.06,E2 -8359.06} C_VEL
LIN {X 0,Y 453.141,Z 452.911,A -85,B 0,C 180,E1 -8360.403,E2 -8360.403} C_VEL
LIN {X 0,Y 452.829,Z 460.255,A -85,B 0,C 180,E1 -8361.747,E2 -8361.747} C_VEL
LIN {X 0,Y 452.669,Z 465.217,A -85,B 0,C 180,E1 -8362.866,E2 -8362.866} C_VEL
LIN {X 0,Y 452.529,Z 470.042,A -85,B 0,C 180,E1 -8364.207,E2 -8364.207} C_VEL
LIN {X 0,Y 452.493,Z 473.736,A -85,B 0,C 180,E1 -8365.546,E2 -8365.546} C_VEL
LIN {X 0,Y 452.492,Z 475.643,A -85,B 0,C 180,E1 -8366.438,E2 -8366.438} C_VEL
LIN {X 0,Y 452.524,Z 477.076,A -85,B 0,C 180,E1 -8367.33,E2 -8367.33} C_VEL
LIN {X 0,Y 452.492,Z 478.729,A -85,B 0,C 180,E1 -8369.11,E2 -8369.11} C_VEL
LIN {X 0,Y 452.471,Z 478.95,A -85,B 0,C 180,E1 -8370,E2 -8370} C_VEL
LIN {X 0,Y 452.492,Z 478.731,A -85,B 0,C 180,E1 -8370.89,E2 -8370.89} C_VEL
LIN {X 0,Y 452.523,Z 477.106,A -85,B 0,C 180,E1 -8372.67,E2 -8372.67} C_VEL
LIN {X 0,Y 452.487,Z 475.667,A -85,B 0,C 180,E1 -8373.561,E2 -8373.561} C_VEL
LIN {X 0,Y 452.548,Z 472.671,A -85,B 0,C 180,E1 -8374.899,E2 -8374.899} C_VEL
LIN {X 0,Y 452.611,Z 468.038,A -85,B 0,C 180,E1 -8376.395,E2 -8376.395} C_VEL
LIN {X 0,Y 452.76,Z 462.333,A -85,B 0,C 180,E1 -8377.805,E2 -8377.805} C_VEL
LIN {X 0,Y 453.042,Z 455.498,A -85,B 0,C 180,E1 -8379.148,E2 -8379.148} C_VEL
LIN {X 0,Y 453.4,Z 446.992,A -85,B 0,C 180,E1 -8380.493,E2 -8380.493} C_VEL
LIN {X 0,Y 453.878,Z 438.225,A -85,B 0,C 180,E1 -8381.611,E2 -8381.611} C_VEL
LIN {X 0,Y 454.447,Z 427.156,A -85,B 0,C 180,E1 -8382.756,E2 -8382.756} C_VEL
LIN {X 0,Y 454.962,Z 416.699,A -85,B 0,C 180,E1 -8383.624,E2 -8383.624} C_VEL
LIN {X 0,Y 455.466,Z 404.672,A -85,B 0,C 180,E1 -8384.406,E2 -8384.406} C_VEL
LIN {X 0,Y 455.971,Z 392.189,A -85,B 0,C 180,E1 -8385.017,E2 -8385.017} C_VEL
LIN {X 0,Y 456.422,Z 379.27,A -85,B 0,C 180,E1 -8385.459,E2 -8385.459} C_VEL
LIN {X 0,Y 456.703,Z 363.997,A -85,B 0,C 180,E1 -8385.764,E2 -8385.764} C_VEL
LIN {X 0,Y 457.292,Z 286.584,A -85,B 0,C 180,E1 -8387.046,E2 -8387.046} C_VEL
LIN {X 0,Y 454.305,Z 266.191,A -85,B 0,C 180,E1 -8387.509,E2 -8387.509} C_VEL
LIN {X 0,Y 455.035,Z 249.856,A -85,B 0,C 180,E1 -8390.333,E2 -8390.333} C_VEL
LIN {X 0,Y 455.884,Z 232.42,A -85,B 0,C 180,E1 -8393.386,E2 -8393.386} C_VEL
LIN {X 0,Y 456.038,Z 225.628,A -85,B 0,C 180,E1 -8394.598,E2 -8394.598} C_VEL
LIN {X 0,Y 453.586,Z 212.986,A -85,B 0,C 180,E1 -8397.04,E2 -8397.04} C_VEL
LIN {X 0,Y 453.461,Z 213.002,A -85,B 0,C 180,E1 -8399.781,E2 -8399.781} C_VEL
LIN {X 0,Y 453.477,Z 212.994,A -85,B 0,C 180,E1 -8403.186,E2 -8403.186} C_VEL
LIN {X 0,Y 453.438,Z 213.002,A -85,B 0,C 180,E1 -8406.296,E2 -8406.296} C_VEL
LIN {X 0,Y 453.47,Z 212.997,A -85,B 0,C 180,E1 -8409.446,E2 -8409.446} C_VEL
LIN {X 0,Y 453.455,Z 213.003,A -85,B 0,C 180,E1 -8411.931,E2 -8411.931} C_VEL
LIN {X 0,Y 453.461,Z 212.999,A -85,B 0,C 180,E1 -8415.468,E2 -8415.468} C_VEL
LIN {X 0,Y 453.451,Z 212.999,A -85,B 0,C 180,E1 -8418.206,E2 -8418.206} C_VEL
LIN {X 0,Y 453.441,Z 212.998,A -85,B 0,C 180,E1 -8420.794,E2 -8420.794} C_VEL
LIN {X 0,Y 453.423,Z 213.004,A -85,B 0,C 180,E1 -8423.914,E2 -8423.914} C_VEL
LIN {X 0,Y 453.447,Z 213,A -85,B 0,C 180,E1 -8427.148,E2 -8427.148} C_VEL
LIN {X 0,Y 453.435,Z 212.999,A -85,B 0,C 180,E1 -8430.265,E2 -8430.265} C_VEL
LIN {X 0,Y 453.466,Z 213.001,A -85,B 0,C 180,E1 -8433.291,E2 -8433.291} C_VEL
LIN {X 0,Y 453.461,Z 212.996,A -85,B 0,C 180,E1 -8436.236,E2 -8436.236} C_VEL
LIN {X 0,Y 453.439,Z 213.003,A -85,B 0,C 180,E1 -8439.115,E2 -8439.115} C_VEL
LIN {X 0,Y 453.465,Z 212.996,A -85,B 0,C 180,E1 -8441.942,E2 -8441.942} C_VEL
LIN {X 0,Y 453.491,Z 212.994,A -85,B 0,C 180,E1 -8444.724,E2 -8444.724} C_VEL
LIN {X 0,Y 453.555,Z 212.988,A -85,B 0,C 180,E1 -8447.471,E2 -8447.471} C_VEL
LIN {X 0,Y 453.543,Z 212.993,A -85,B 0,C 180,E1 -8451.085,E2 -8451.085} C_VEL
LIN {X 0,Y 453.615,Z 212.977,A -85,B 0,C 180,E1 -8453.774,E2 -8453.774} C_VEL
LIN {X 0,Y 453.691,Z 212.97,A -85,B 0,C 180,E1 -8457.336,E2 -8457.336} C_VEL
LIN {X 0,Y 453.767,Z 212.957,A -85,B 0,C 180,E1 -8460,E2 -8460} C_VEL
LIN {X 0,Y 453.693,Z 212.972,A -85,B 0,C 180,E1 -8462.663,E2 -8462.663} C_VEL
LIN {X 0,Y 453.642,Z 212.974,A -85,B 0,C 180,E1 -8466.225,E2 -8466.225} C_VEL
LIN {X 0,Y 453.544,Z 212.991,A -85,B 0,C 180,E1 -8468.914,E2 -8468.914} C_VEL
LIN {X 0,Y 453.554,Z 212.99,A -85,B 0,C 180,E1 -8472.552,E2 -8472.552} C_VEL
LIN {X 0,Y 453.509,Z 212.992,A -85,B 0,C 180,E1 -8476.197,E2 -8476.197} C_VEL
LIN {X 0,Y 453.475,Z 212.996,A -85,B 0,C 180,E1 -8479.043,E2 -8479.043} C_VEL
LIN {X 0,Y 453.482,Z 212.994,A -85,B 0,C 180,E1 -8481.836,E2 -8481.836} C_VEL
LIN {X 0,Y 453.488,Z 212.996,A -85,B 0,C 180,E1 -8484.736,E2 -8484.736} C_VEL
LIN {X 0,Y 453.497,Z 212.994,A -85,B 0,C 180,E1 -8487.963,E2 -8487.963} C_VEL
LIN {X 0,Y 453.444,Z 213,A -85,B 0,C 180,E1 -8490.762,E2 -8490.762} C_VEL
LIN {X 0,Y 453.44,Z 213.001,A -85,B 0,C 180,E1 -8493.915,E2 -8493.915} C_VEL
LIN {X 0,Y 453.437,Z 212.998,A -85,B 0,C 180,E1 -8497.191,E2 -8497.191} C_VEL
LIN {X 0,Y 453.505,Z 212.991,A -85,B 0,C 180,E1 -8499.448,E2 -8499.448} C_VEL
LIN {X 0,Y 453.462,Z 212.995,A -85,B 0,C 180,E1 -8502.995,E2 -8502.995} C_VEL
LIN {X 0,Y 453.438,Z 213.003,A -85,B 0,C 180,E1 -8505.782,E2 -8505.782} C_VEL
LIN {X 0,Y 453.493,Z 212.993,A -85,B 0,C 180,E1 -8509.409,E2 -8509.409} C_VEL
LIN {X 0,Y 453.454,Z 213,A -85,B 0,C 180,E1 -8512.226,E2 -8512.226} C_VEL
LIN {X 0,Y 453.47,Z 212.995,A -85,B 0,C 180,E1 -8515.225,E2 -8515.225} C_VEL
LIN {X 0,Y 453.452,Z 212.997,A -85,B 0,C 180,E1 -8518.477,E2 -8518.477} C_VEL
LIN {X 0,Y 453.501,Z 212.993,A -85,B 0,C 180,E1 -8521.291,E2 -8521.291} C_VEL
LIN {X 0,Y 453.514,Z 212.99,A -85,B 0,C 180,E1 -8524.287,E2 -8524.287} C_VEL
LIN {X 0,Y 453.471,Z 212.997,A -85,B 0,C 180,E1 -8527.206,E2 -8527.206} C_VEL
LIN {X 0,Y 453.497,Z 212.993,A -85,B 0,C 180,E1 -8530.068,E2 -8530.068} C_VEL
LIN {X 0,Y 453.5,Z 212.992,A -85,B 0,C 180,E1 -8532.878,E2 -8532.878} C_VEL
LIN {X 0,Y 453.511,Z 212.995,A -85,B 0,C 180,E1 -8535.645,E2 -8535.645} C_VEL
LIN {X 0,Y 453.556,Z 212.984,A -85,B 0,C 180,E1 -8538.38,E2 -8538.38} C_VEL
LIN {X 0,Y 453.65,Z 212.973,A -85,B 0,C 180,E1 -8541.986,E2 -8541.986} C_VEL
LIN {X 0,Y 453.627,Z 212.976,A -85,B 0,C 180,E1 -8543.136,E2 -8543.136} C_VEL
LIN {X 0,Y 452.946,Z 213.063,A -85,B 0,C 180,E1 -8543.877,E2 -8543.877} C_VEL
LIN {X 0,Y 450.001,Z 213.431,A -85,B 0,C 180,E1 -8545.078,E2 -8545.078} C_VEL
LIN {X 0,Y 447.582,Z 213.729,A -85,B 0,C 180,E1 -8546.048,E2 -8546.048} C_VEL
LIN {X 0,Y 446.65,Z 213.846,A -85,B 0,C 180,E1 -8546.798,E2 -8546.798} C_VEL
LIN {X 0,Y 446.633,Z 213.85,A -85,B 0,C 180,E1 -8547.051,E2 -8547.051} C_VEL
LIN {X 0,Y 446.791,Z 213.827,A -85,B 0,C 180,E1 -8550,E2 -8550} C_VEL
LIN {X 0,Y 446.708,Z 213.839,A -85,B 0,C 180,E1 -8552.705,E2 -8552.705} C_VEL
LIN {X 0,Y 446.628,Z 213.847,A -85,B 0,C 180,E1 -8556.323,E2 -8556.323} C_VEL
LIN {X 0,Y 446.536,Z 213.866,A -85,B 0,C 180,E1 -8559.054,E2 -8559.054} C_VEL
LIN {X 0,Y 446.518,Z 213.865,A -85,B 0,C 180,E1 -8562.728,E2 -8562.728} C_VEL
LIN {X 0,Y 446.491,Z 213.865,A -85,B 0,C 180,E1 -8566.226,E2 -8566.226} C_VEL
LIN {X 0,Y 446.463,Z 213.87,A -85,B 0,C 180,E1 -8569.301,E2 -8569.301} C_VEL
LIN {X 0,Y 446.41,Z 213.875,A -85,B 0,C 180,E1 -8572.198,E2 -8572.198} C_VEL
LIN {X 0,Y 446.448,Z 213.874,A -85,B 0,C 180,E1 -8575.15,E2 -8575.15} C_VEL
LIN {X 0,Y 446.472,Z 213.872,A -85,B 0,C 180,E1 -8578.176,E2 -8578.176} C_VEL
LIN {X 0,Y 446.521,Z 213.95,A -85,B 0,C 180,E1 -8579.459,E2 -8579.459} C_VEL
LIN {X 0,Y 447.698,Z 220.419,A -85,B 0,C 180,E1 -8580.934,E2 -8580.934} C_VEL
LIN {X 0,Y 447.611,Z 226.893,A -85,B 0,C 180,E1 -8582.321,E2 -8582.321} C_VEL
LIN {X 0,Y 450.829,Z 242.676,A -85,B 0,C 180,E1 -8582.72,E2 -8582.72} C_VEL
LIN {X 0,Y 449.822,Z 333.973,A -85,B 0,C 180,E1 -8584.273,E2 -8584.273} C_VEL
LIN {X 0,Y 449.443,Z 347.387,A -85,B 0,C 180,E1 -8584.679,E2 -8584.679} C_VEL
LIN {X 0,Y 449.166,Z 359.656,A -85,B 0,C 180,E1 -8585.234,E2 -8585.234} C_VEL
LIN {X 0,Y 448.687,Z 371.1,A -85,B 0,C 180,E1 -8585.922,E2 -8585.922} C_VEL
LIN {X 0,Y 448.191,Z 381.492,A -85,B 0,C 180,E1 -8586.719,E2 -8586.719} C_VEL
LIN {X 0,Y 447.659,Z 392.262,A -85,B 0,C 180,E1 -8587.75,E2 -8587.75} C_VEL
LIN {X 0,Y 447.096,Z 402.407,A -85,B 0,C 180,E1 -8588.954,E2 -8588.954} C_VEL
LIN {X 0,Y 446.627,Z 411.713,A -85,B 0,C 180,E1 -8590.35,E2 -8590.35} C_VEL
LIN {X 0,Y 446.133,Z 419.524,A -85,B 0,C 180,E1 -8591.814,E2 -8591.814} C_VEL
LIN {X 0,Y 445.934,Z 424.882,A -85,B 0,C 180,E1 -8593.079,E2 -8593.079} C_VEL
LIN {X 0,Y 445.739,Z 429.23,A -85,B 0,C 180,E1 -8594.362,E2 -8594.362} C_VEL
LIN {X 0,Y 445.506,Z 433.445,A -85,B 0,C 180,E1 -8596.044,E2 -8596.044} C_VEL
LIN {X 0,Y 445.38,Z 436.341,A -85,B 0,C 180,E1 -8597.865,E2 -8597.865} C_VEL
LIN {X 0,Y 445.302,Z 437.53,A -85,B 0,C 180,E1 -8599.678,E2 -8599.678} C_VEL
LIN {X 0,Y 445.307,Z 437.478,A -85,B 0,C 180,E1 -8600.855,E2 -8600.855} C_VEL
LIN {X 0,Y 445.32,Z 436.652,A -85,B 0,C 180,E1 -8602.093,E2 -8602.093} C_VEL
LIN {X 0,Y 445.437,Z 434.69,A -85,B 0,C 180,E1 -8603.57,E2 -8603.57} C_VEL
LIN {X 0,Y 445.607,Z 431.494,A -85,B 0,C 180,E1 -8605.089,E2 -8605.089} C_VEL
LIN {X 0,Y 445.876,Z 426.824,A -85,B 0,C 180,E1 -8606.648,E2 -8606.648} C_VEL
LIN {X 0,Y 446.236,Z 420.431,A -85,B 0,C 180,E1 -8608.253,E2 -8608.253} C_VEL
LIN {X 0,Y 446.602,Z 414.126,A -85,B 0,C 180,E1 -8609.503,E2 -8609.503} C_VEL
LIN {X 0,Y 447.118,Z 405.786,A -85,B 0,C 180,E1 -8610.839,E2 -8610.839} C_VEL
LIN {X 0,Y 447.662,Z 396.581,A -85,B 0,C 180,E1 -8612.03,E2 -8612.03} C_VEL
LIN {X 0,Y 448.116,Z 386.843,A -85,B 0,C 180,E1 -8613.06,E2 -8613.06} C_VEL
LIN {X 0,Y 448.774,Z 375.814,A -85,B 0,C 180,E1 -8613.993,E2 -8613.993} C_VEL
LIN {X 0,Y 449.314,Z 364.02,A -85,B 0,C 180,E1 -8614.772,E2 -8614.772} C_VEL
LIN {X 0,Y 449.775,Z 351.065,A -85,B 0,C 180,E1 -8615.416,E2 -8615.416} C_VEL
LIN {X 0,Y 450.042,Z 337.983,A -85,B 0,C 180,E1 -8615.861,E2 -8615.861} C_VEL
LIN {X 0,Y 450.291,Z 319.139,A -85,B 0,C 180,E1 -8616.227,E2 -8616.227} C_VEL
LIN {X 0,Y 451.226,Z 242.796,A -85,B 0,C 180,E1 -8617.538,E2 -8617.538} C_VEL
LIN {X 0,Y 447.878,Z 226.992,A -85,B 0,C 180,E1 -8617.998,E2 -8617.998} C_VEL
LIN {X 0,Y 447.763,Z 220.142,A -85,B 0,C 180,E1 -8619.32,E2 -8619.32} C_VEL
LIN {X 0,Y 446.481,Z 213.872,A -85,B 0,C 180,E1 -8620.638,E2 -8620.638} C_VEL
LIN {X 0,Y 446.473,Z 213.872,A -85,B 0,C 180,E1 -8623.761,E2 -8623.761} C_VEL
LIN {X 0,Y 446.507,Z 213.873,A -85,B 0,C 180,E1 -8627.361,E2 -8627.361} C_VEL
LIN {X 0,Y 446.492,Z 213.871,A -85,B 0,C 180,E1 -8630.944,E2 -8630.944} C_VEL
LIN {X 0,Y 446.611,Z 213.853,A -85,B 0,C 180,E1 -8633.676,E2 -8633.676} C_VEL
LIN {X 0,Y 446.641,Z 213.853,A -85,B 0,C 180,E1 -8637.295,E2 -8637.295} C_VEL
LIN {X 0,Y 446.739,Z 213.835,A -85,B 0,C 180,E1 -8640,E2 -8640} C_VEL
LIN {X 0,Y 446.64,Z 213.851,A -85,B 0,C 180,E1 -8642.706,E2 -8642.706} C_VEL
LIN {X 0,Y 446.586,Z 213.852,A -85,B 0,C 180,E1 -8646.325,E2 -8646.325} C_VEL
LIN {X 0,Y 446.491,Z 213.869,A -85,B 0,C 180,E1 -8649.057,E2 -8649.057} C_VEL
LIN {X 0,Y 446.488,Z 213.87,A -85,B 0,C 180,E1 -8652.731,E2 -8652.731} C_VEL
LIN {X 0,Y 446.451,Z 213.874,A -85,B 0,C 180,E1 -8656.461,E2 -8656.461} C_VEL
LIN {X 0,Y 446.426,Z 213.873,A -85,B 0,C 180,E1 -8659.305,E2 -8659.305} C_VEL
LIN {X 0,Y 446.378,Z 213.882,A -85,B 0,C 180,E1 -8662.202,E2 -8662.202} C_VEL
LIN {X 0,Y 446.417,Z 213.876,A -85,B 0,C 180,E1 -8665.155,E2 -8665.155} C_VEL
LIN {X 0,Y 446.448,Z 213.873,A -85,B 0,C 180,E1 -8668.181,E2 -8668.181} C_VEL
LIN {X 0,Y 446.383,Z 213.879,A -85,B 0,C 180,E1 -8671.777,E2 -8671.777} C_VEL
LIN {X 0,Y 446.397,Z 213.88,A -85,B 0,C 180,E1 -8674.526,E2 -8674.526} C_VEL
LIN {X 0,Y 446.383,Z 213.882,A -85,B 0,C 180,E1 -8678.082,E2 -8678.082} C_VEL
LIN {X 0,Y 446.398,Z 213.877,A -85,B 0,C 180,E1 -8680.921,E2 -8680.921} C_VEL
LIN {X 0,Y 446.372,Z 213.881,A -85,B 0,C 180,E1 -8683.85,E2 -8683.85} C_VEL
LIN {X 0,Y 446.373,Z 213.884,A -85,B 0,C 180,E1 -8686.407,E2 -8686.407} C_VEL
LIN {X 0,Y 446.407,Z 213.876,A -85,B 0,C 180,E1 -8689.086,E2 -8689.086} C_VEL
LIN {X 0,Y 446.392,Z 213.883,A -85,B 0,C 180,E1 -8692.124,E2 -8692.124} C_VEL
LIN {X 0,Y 446.416,Z 213.876,A -85,B 0,C 180,E1 -8695.48,E2 -8695.48} C_VEL
LIN {X 0,Y 446.404,Z 213.879,A -85,B 0,C 180,E1 -8698.703,E2 -8698.703} C_VEL
LIN {X 0,Y 446.477,Z 213.875,A -85,B 0,C 180,E1 -8701.824,E2 -8701.824} C_VEL
LIN {X 0,Y 446.525,Z 214.02,A -85,B 0,C 180,E1 -8703.102,E2 -8703.102} C_VEL
LIN {X 0,Y 448.49,Z 223.817,A -85,B 0,C 180,E1 -8704.972,E2 -8704.972} C_VEL
LIN {X 0,Y 449.009,Z 227.432,A -85,B 0,C 180,E1 -8705.642,E2 -8705.642} C_VEL
LIN {X 0,Y 448.333,Z 241.856,A -85,B 0,C 180,E1 -8708.145,E2 -8708.145} C_VEL
LIN {X 0,Y 447.468,Z 262.524,A -85,B 0,C 180,E1 -8711.694,E2 -8711.694} C_VEL
LIN {X 0,Y 447.371,Z 264.523,A -85,B 0,C 180,E1 -8712.034,E2 -8712.034} C_VEL
LIN {X 0,Y 450.845,Z 288.226,A -85,B 0,C 180,E1 -8712.618,E2 -8712.618} C_VEL
LIN {X 0,Y 449.932,Z 374.338,A -85,B 0,C 180,E1 -8714.109,E2 -8714.109} C_VEL
LIN {X 0,Y 449.467,Z 387.221,A -85,B 0,C 180,E1 -8714.499,E2 -8714.499} C_VEL
LIN {X 0,Y 448.85,Z 400.362,A -85,B 0,C 180,E1 -8715.087,E2 -8715.087} C_VEL
LIN {X 0,Y 448.279,Z 412.281,A -85,B 0,C 180,E1 -8715.822,E2 -8715.822} C_VEL
LIN {X 0,Y 447.677,Z 423.888,A -85,B 0,C 180,E1 -8716.738,E2 -8716.738} C_VEL
LIN {X 0,Y 447.106,Z 434.168,A -85,B 0,C 180,E1 -8717.75,E2 -8717.75} C_VEL
LIN {X 0,Y 446.598,Z 443.513,A -85,B 0,C 180,E1 -8718.886,E2 -8718.886} C_VEL
LIN {X 0,Y 446.111,Z 452.612,A -85,B 0,C 180,E1 -8720.251,E2 -8720.251} C_VEL
LIN {X 0,Y 445.77,Z 459.949,A -85,B 0,C 180,E1 -8721.615,E2 -8721.615} C_VEL
LIN {X 0,Y 445.597,Z 464.906,A -85,B 0,C 180,E1 -8722.752,E2 -8722.752} C_VEL
LIN {X 0,Y 445.444,Z 469.32,A -85,B 0,C 180,E1 -8723.988,E2 -8723.988} C_VEL
LIN {X 0,Y 445.417,Z 473.422,A -85,B 0,C 180,E1 -8725.476,E2 -8725.476} C_VEL
LIN {X 0,Y 445.392,Z 475.325,A -85,B 0,C 180,E1 -8726.382,E2 -8726.382} C_VEL
LIN {X 0,Y 445.448,Z 476.756,A -85,B 0,C 180,E1 -8727.287,E2 -8727.287} C_VEL
LIN {X 0,Y 445.398,Z 478.406,A -85,B 0,C 180,E1 -8729.096,E2 -8729.096} C_VEL
LIN {X 0,Y 445.407,Z 478.622,A -85,B 0,C 180,E1 -8730,E2 -8730} C_VEL
LIN {X 0,Y 445.398,Z 478.397,A -85,B 0,C 180,E1 -8730.904,E2 -8730.904} C_VEL
LIN {X 0,Y 445.446,Z 476.763,A -85,B 0,C 180,E1 -8732.713,E2 -8732.713} C_VEL
LIN {X 0,Y 445.388,Z 475.312,A -85,B 0,C 180,E1 -8733.618,E2 -8733.618} C_VEL
LIN {X 0,Y 445.478,Z 472.306,A -85,B 0,C 180,E1 -8734.977,E2 -8734.977} C_VEL
LIN {X 0,Y 445.53,Z 468.059,A -85,B 0,C 180,E1 -8736.385,E2 -8736.385} C_VEL
LIN {X 0,Y 445.702,Z 461.932,A -85,B 0,C 180,E1 -8737.93,E2 -8737.93} C_VEL
LIN {X 0,Y 445.979,Z 455.075,A -85,B 0,C 180,E1 -8739.294,E2 -8739.294} C_VEL
LIN {X 0,Y 446.36,Z 446.532,A -85,B 0,C 180,E1 -8740.66,E2 -8740.66} C_VEL
LIN {X 0,Y 446.869,Z 437.735,A -85,B 0,C 180,E1 -8741.796,E2 -8741.796} C_VEL
LIN {X 0,Y 447.418,Z 427.639,A -85,B 0,C 180,E1 -8742.862,E2 -8742.862} C_VEL
LIN {X 0,Y 448.025,Z 416.111,A -85,B 0,C 180,E1 -8743.839,E2 -8743.839} C_VEL
LIN {X 0,Y 448.567,Z 403.999,A -85,B 0,C 180,E1 -8744.632,E2 -8744.632} C_VEL
LIN {X 0,Y 449.098,Z 391.407,A -85,B 0,C 180,E1 -8745.252,E2 -8745.252} C_VEL
LIN {X 0,Y 449.576,Z 378.152,A -85,B 0,C 180,E1 -8745.7,E2 -8745.7} C_VEL
LIN {X 0,Y 449.901,Z 360.796,A -85,B 0,C 180,E1 -8746.038,E2 -8746.038} C_VEL
LIN {X 0,Y 450.412,Z 287.002,A -85,B 0,C 180,E1 -8747.286,E2 -8747.286} C_VEL
LIN {X 0,Y 447.304,Z 265.786,A -85,B 0,C 180,E1 -8747.792,E2 -8747.792} C_VEL
LIN {X 0,Y 448.07,Z 249.465,A -85,B 0,C 180,E1 -8750.663,E2 -8750.663} C_VEL
LIN {X 0,Y 448.95,Z 233.38,A -85,B 0,C 180,E1 -8753.524,E2 -8753.524} C_VEL
LIN {X 0,Y 449.208,Z 228.356,A -85,B 0,C 180,E1 -8754.426,E2 -8754.426} C_VEL
LIN {X 0,Y 447.711,Z 219.814,A -85,B 0,C 180,E1 -8756.071,E2 -8756.071} C_VEL
LIN {X 0,Y 446.532,Z 213.865,A -85,B 0,C 180,E1 -8757.281,E2 -8757.281} C_VEL
LIN {X 0,Y 446.416,Z 213.88,A -85,B 0,C 180,E1 -8760.247,E2 -8760.247} C_VEL
LIN {X 0,Y 446.432,Z 213.873,A -85,B 0,C 180,E1 -8763.45,E2 -8763.45} C_VEL
LIN {X 0,Y 446.386,Z 213.877,A -85,B 0,C 180,E1 -8766.742,E2 -8766.742} C_VEL
LIN {X 0,Y 446.424,Z 213.876,A -85,B 0,C 180,E1 -8770.195,E2 -8770.195} C_VEL
LIN {X 0,Y 446.406,Z 213.875,A -85,B 0,C 180,E1 -8772.601,E2 -8772.601} C_VEL
LIN {X 0,Y 446.428,Z 213.872,A -85,B 0,C 180,E1 -8775.1,E2 -8775.1} C_VEL
LIN {X 0,Y 446.4,Z 213.875,A -85,B 0,C 180,E1 -8778.605,E2 -8778.605} C_VEL
LIN {X 0,Y 446.382,Z 213.882,A -85,B 0,C 180,E1 -8781.918,E2 -8781.918} C_VEL
LIN {X 0,Y 446.396,Z 213.882,A -85,B 0,C 180,E1 -8785.474,E2 -8785.474} C_VEL
LIN {X 0,Y 446.378,Z 213.878,A -85,B 0,C 180,E1 -8788.696,E2 -8788.696} C_VEL
LIN {X 0,Y 446.447,Z 213.873,A -85,B 0,C 180,E1 -8791.818,E2 -8791.818} C_VEL
LIN {X 0,Y 446.416,Z 213.875,A -85,B 0,C 180,E1 -8794.845,E2 -8794.845} C_VEL
LIN {X 0,Y 446.406,Z 213.874,A -85,B 0,C 180,E1 -8798.243,E2 -8798.243} C_VEL
LIN {X 0,Y 446.412,Z 213.877,A -85,B 0,C 180,E1 -8801.647,E2 -8801.647} C_VEL
LIN {X 0,Y 446.46,Z 213.868,A -85,B 0,C 180,E1 -8804.478,E2 -8804.478} C_VEL
LIN {X 0,Y 446.492,Z 213.864,A -85,B 0,C 180,E1 -8808.192,E2 -8808.192} C_VEL
LIN {X 0,Y 446.551,Z 213.857,A -85,B 0,C 180,E1 -8811.857,E2 -8811.857} C_VEL
LIN {X 0,Y 446.588,Z 213.854,A -85,B 0,C 180,E1 -8814.582,E2 -8814.582} C_VEL
LIN {X 0,Y 446.612,Z 213.849,A -85,B 0,C 180,E1 -8818.196,E2 -8818.196} C_VEL
LIN {X 0,Y 446.738,Z 213.833,A -85,B 0,C 180,E1 -8820,E2 -8820} C_VEL
LIN {X 0,Y 446.64,Z 213.851,A -85,B 0,C 180,E1 -8822.705,E2 -8822.705} C_VEL
LIN {X 0,Y 446.61,Z 213.851,A -85,B 0,C 180,E1 -8826.324,E2 -8826.324} C_VEL
LIN {X 0,Y 446.49,Z 213.868,A -85,B 0,C 180,E1 -8829.056,E2 -8829.056} C_VEL
LIN {X 0,Y 446.487,Z 213.872,A -85,B 0,C 180,E1 -8832.73,E2 -8832.73} C_VEL
LIN {X 0,Y 446.449,Z 213.875,A -85,B 0,C 180,E1 -8836.46,E2 -8836.46} C_VEL
LIN {X 0,Y 446.429,Z 213.872,A -85,B 0,C 180,E1 -8839.305,E2 -8839.305} C_VEL
LIN {X 0,Y 446.421,Z 213.876,A -85,B 0,C 180,E1 -8842.199,E2 -8842.199} C_VEL
LIN {X 0,Y 446.432,Z 213.872,A -85,B 0,C 180,E1 -8845.153,E2 -8845.153} C_VEL
LIN {X 0,Y 446.445,Z 213.875,A -85,B 0,C 180,E1 -8848.181,E2 -8848.181} C_VEL
LIN {X 0,Y 446.379,Z 213.878,A -85,B 0,C 180,E1 -8851.303,E2 -8851.303} C_VEL
LIN {X 0,Y 446.394,Z 213.88,A -85,B 0,C 180,E1 -8854.526,E2 -8854.526} C_VEL
LIN {X 0,Y 446.406,Z 213.881,A -85,B 0,C 180,E1 -8858.086,E2 -8858.086} C_VEL
LIN {X 0,Y 446.416,Z 213.873,A -85,B 0,C 180,E1 -8860.923,E2 -8860.923} C_VEL
LIN {X 0,Y 446.416,Z 213.878,A -85,B 0,C 180,E1 -8863.844,E2 -8863.844} C_VEL
LIN {X 0,Y 446.372,Z 213.882,A -85,B 0,C 180,E1 -8866.407,E2 -8866.407} C_VEL
LIN {X 0,Y 446.445,Z 213.875,A -85,B 0,C 180,E1 -8869.808,E2 -8869.808} C_VEL
LIN {X 0,Y 446.41,Z 213.879,A -85,B 0,C 180,E1 -8872.126,E2 -8872.126} C_VEL
LIN {X 0,Y 446.412,Z 213.877,A -85,B 0,C 180,E1 -8875.48,E2 -8875.48} C_VEL
LIN {X 0,Y 446.404,Z 213.875,A -85,B 0,C 180,E1 -8878.703,E2 -8878.703} C_VEL
LIN {X 0,Y 446.472,Z 213.873,A -85,B 0,C 180,E1 -8881.824,E2 -8881.824} C_VEL
LIN {X 0,Y 446.447,Z 213.869,A -85,B 0,C 180,E1 -8884.85,E2 -8884.85} C_VEL
LIN {X 0,Y 446.44,Z 213.871,A -85,B 0,C 180,E1 -8888.247,E2 -8888.247} C_VEL
LIN {X 0,Y 446.451,Z 213.875,A -85,B 0,C 180,E1 -8891.651,E2 -8891.651} C_VEL
LIN {X 0,Y 446.503,Z 213.862,A -85,B 0,C 180,E1 -8894.481,E2 -8894.481} C_VEL
LIN {X 0,Y 446.514,Z 213.861,A -85,B 0,C 180,E1 -8898.194,E2 -8898.194} C_VEL
LIN {X 0,Y 446.598,Z 213.852,A -85,B 0,C 180,E1 -8901.859,E2 -8901.859} C_VEL
LIN {X 0,Y 446.641,Z 213.846,A -85,B 0,C 180,E1 -8904.583,E2 -8904.583} C_VEL
LIN {X 0,Y 446.633,Z 213.85,A -85,B 0,C 180,E1 -8907.051,E2 -8907.051} C_VEL
LIN {X 0,Y 446.433,Z 213.88,A -85,B 0,C 180,E1 -8907.555,E2 -8907.555} C_VEL
LIN {X 0,Y 445.163,Z 214.043,A -85,B 0,C 180,E1 -8908.298,E2 -8908.298} C_VEL
LIN {X 0,Y 440.784,Z 214.586,A -85,B 0,C 180,E1 -8910.014,E2 -8910.014} C_VEL
LIN {X 0,Y 439.697,Z 214.715,A -85,B 0,C 180,E1 -8910.777,E2 -8910.777} C_VEL
LIN {X 0,Y 439.607,Z 214.724,A -85,B 0,C 180,E1 -8911.036,E2 -8911.036} C_VEL
LIN {X 0,Y 439.654,Z 214.718,A -85,B 0,C 180,E1 -8912.748,E2 -8912.748} C_VEL
LIN {X 0,Y 439.598,Z 214.723,A -85,B 0,C 180,E1 -8916.425,E2 -8916.425} C_VEL
LIN {X 0,Y 439.497,Z 214.74,A -85,B 0,C 180,E1 -8919.201,E2 -8919.201} C_VEL
LIN {X 0,Y 439.462,Z 214.747,A -85,B 0,C 180,E1 -8922.936,E2 -8922.936} C_VEL
LIN {X 0,Y 439.442,Z 214.743,A -85,B 0,C 180,E1 -8926.347,E2 -8926.347} C_VEL
LIN {X 0,Y 439.396,Z 214.748,A -85,B 0,C 180,E1 -8929.624,E2 -8929.624} C_VEL
LIN {X 0,Y 439.356,Z 214.758,A -85,B 0,C 180,E1 -8932.573,E2 -8932.573} C_VEL
LIN {X 0,Y 439.395,Z 214.751,A -85,B 0,C 180,E1 -8935.583,E2 -8935.583} C_VEL
LIN {X 0,Y 439.433,Z 214.751,A -85,B 0,C 180,E1 -8938.669,E2 -8938.669} C_VEL
LIN {X 0,Y 439.494,Z 214.876,A -85,B 0,C 180,E1 -8939.286,E2 -8939.286} C_VEL
LIN {X 0,Y 440.765,Z 222.037,A -85,B 0,C 180,E1 -8940.942,E2 -8940.942} C_VEL
LIN {X 0,Y 440.684,Z 227.367,A -85,B 0,C 180,E1 -8942.055,E2 -8942.055} C_VEL
LIN {X 0,Y 444.052,Z 244.329,A -85,B 0,C 180,E1 -8942.492,E2 -8942.492} C_VEL
LIN {X 0,Y 442.956,Z 333.931,A -85,B 0,C 180,E1 -8944.039,E2 -8944.039} C_VEL
LIN {X 0,Y 442.606,Z 347.025,A -85,B 0,C 180,E1 -8944.437,E2 -8944.437} C_VEL
LIN {X 0,Y 442.285,Z 360.017,A -85,B 0,C 180,E1 -8945.028,E2 -8945.028} C_VEL
LIN {X 0,Y 441.751,Z 372.046,A -85,B 0,C 180,E1 -8945.77,E2 -8945.77} C_VEL
LIN {X 0,Y 441.15,Z 383.471,A -85,B 0,C 180,E1 -8946.68,E2 -8946.68} C_VEL
LIN {X 0,Y 440.595,Z 394.068,A -85,B 0,C 180,E1 -8947.739,E2 -8947.739} C_VEL
LIN {X 0,Y 440.008,Z 403.882,A -85,B 0,C 180,E1 -8948.964,E2 -8948.964} C_VEL
LIN {X 0,Y 439.546,Z 413.083,A -85,B 0,C 180,E1 -8950.397,E2 -8950.397} C_VEL
LIN {X 0,Y 439.091,Z 419.841,A -85,B 0,C 180,E1 -8951.705,E2 -8951.705} C_VEL
LIN {X 0,Y 438.886,Z 425.249,A -85,B 0,C 180,E1 -8953.004,E2 -8953.004} C_VEL
LIN {X 0,Y 438.646,Z 429.831,A -85,B 0,C 180,E1 -8954.388,E2 -8954.388} C_VEL
LIN {X 0,Y 438.465,Z 433.147,A -85,B 0,C 180,E1 -8955.695,E2 -8955.695} C_VEL
LIN {X 0,Y 438.39,Z 434.598,A -85,B 0,C 180,E1 -8956.422,E2 -8956.422} C_VEL
LIN {X 0,Y 438.303,Z 436.437,A -85,B 0,C 180,E1 -8957.666,E2 -8957.666} C_VEL
LIN {X 0,Y 438.266,Z 437.537,A -85,B 0,C 180,E1 -8958.904,E2 -8958.904} C_VEL
LIN {X 0,Y 438.206,Z 437.908,A -85,B 0,C 180,E1 -8960.331,E2 -8960.331} C_VEL
LIN {X 0,Y 438.215,Z 437.282,A -85,B 0,C 180,E1 -8961.791,E2 -8961.791} C_VEL
LIN {X 0,Y 438.375,Z 435.061,A -85,B 0,C 180,E1 -8963.617,E2 -8963.617} C_VEL
LIN {X 0,Y 438.563,Z 431.381,A -85,B 0,C 180,E1 -8965.354,E2 -8965.354} C_VEL
LIN {X 0,Y 438.868,Z 426.313,A -85,B 0,C 180,E1 -8967.012,E2 -8967.012} C_VEL
LIN {X 0,Y 439.209,Z 420.775,A -85,B 0,C 180,E1 -8968.396,E2 -8968.396} C_VEL
LIN {X 0,Y 439.628,Z 414.422,A -85,B 0,C 180,E1 -8969.673,E2 -8969.673} C_VEL
LIN {X 0,Y 440.079,Z 407.289,A -85,B 0,C 180,E1 -8970.852,E2 -8970.852} C_VEL
LIN {X 0,Y 440.631,Z 398.354,A -85,B 0,C 180,E1 -8972.062,E2 -8972.062} C_VEL
LIN {X 0,Y 441.212,Z 387.646,A -85,B 0,C 180,E1 -8973.23,E2 -8973.23} C_VEL
LIN {X 0,Y 441.894,Z 376.597,A -85,B 0,C 180,E1 -8974.191,E2 -8974.191} C_VEL
LIN {X 0,Y 442.465,Z 364.817,A -85,B 0,C 180,E1 -8974.99,E2 -8974.99} C_VEL
LIN {X 0,Y 442.955,Z 352.173,A -85,B 0,C 180,E1 -8975.637,E2 -8975.637} C_VEL
LIN {X 0,Y 443.276,Z 339.552,A -85,B 0,C 180,E1 -8976.091,E2 -8976.091} C_VEL
LIN {X 0,Y 443.497,Z 324.315,A -85,B 0,C 180,E1 -8976.414,E2 -8976.414} C_VEL
LIN {X 0,Y 444.507,Z 243.837,A -85,B 0,C 180,E1 -8977.823,E2 -8977.823} C_VEL
LIN {X 0,Y 440.979,Z 227.434,A -85,B 0,C 180,E1 -8978.295,E2 -8978.295} C_VEL
LIN {X 0,Y 440.825,Z 221.466,A -85,B 0,C 180,E1 -8979.468,E2 -8979.468} C_VEL
LIN {X 0,Y 439.441,Z 214.749,A -85,B 0,C 180,E1 -8980.912,E2 -8980.912} C_VEL
LIN {X 0,Y 439.428,Z 214.749,A -85,B 0,C 180,E1 -8984.224,E2 -8984.224} C_VEL
LIN {X 0,Y 439.466,Z 214.747,A -85,B 0,C 180,E1 -8988.001,E2 -8988.001} C_VEL
LIN {X 0,Y 439.501,Z 214.74,A -85,B 0,C 180,E1 -8991.726,E2 -8991.726} C_VEL
LIN {X 0,Y 439.58,Z 214.728,A -85,B 0,C 180,E1 -8994.496,E2 -8994.496} C_VEL
LIN {X 0,Y 439.583,Z 214.727,A -85,B 0,C 180,E1 -8998.168,E2 -8998.168} C_VEL
LIN {X 0,Y 439.71,Z 214.711,A -85,B 0,C 180,E1 -9000,E2 -9000} C_VEL
LIN {X 0,Y 439.59,Z 214.73,A -85,B 0,C 180,E1 -9002.749,E2 -9002.749} C_VEL
LIN {X 0,Y 439.562,Z 214.728,A -85,B 0,C 180,E1 -9006.426,E2 -9006.426} C_VEL
LIN {X 0,Y 439.454,Z 214.746,A -85,B 0,C 180,E1 -9009.203,E2 -9009.203} C_VEL
LIN {X 0,Y 439.459,Z 214.746,A -85,B 0,C 180,E1 -9012.728,E2 -9012.728} C_VEL
LIN {X 0,Y 439.416,Z 214.749,A -85,B 0,C 180,E1 -9016.356,E2 -9016.356} C_VEL
LIN {X 0,Y 439.359,Z 214.753,A -85,B 0,C 180,E1 -9019.629,E2 -9019.629} C_VEL
LIN {X 0,Y 439.325,Z 214.763,A -85,B 0,C 180,E1 -9022.578,E2 -9022.578} C_VEL
LIN {X 0,Y 439.366,Z 214.752,A -85,B 0,C 180,E1 -9025.588,E2 -9025.588} C_VEL
LIN {X 0,Y 439.38,Z 214.753,A -85,B 0,C 180,E1 -9028.676,E2 -9028.676} C_VEL
LIN {X 0,Y 439.334,Z 214.759,A -85,B 0,C 180,E1 -9032.033,E2 -9032.033} C_VEL
LIN {X 0,Y 439.363,Z 214.75,A -85,B 0,C 180,E1 -9035.343,E2 -9035.343} C_VEL
LIN {X 0,Y 439.341,Z 214.76,A -85,B 0,C 180,E1 -9038.6,E2 -9038.6} C_VEL
LIN {X 0,Y 439.359,Z 214.753,A -85,B 0,C 180,E1 -9041.26,E2 -9041.26} C_VEL
LIN {X 0,Y 439.375,Z 214.752,A -85,B 0,C 180,E1 -9044.733,E2 -9044.733} C_VEL
LIN {X 0,Y 439.375,Z 214.754,A -85,B 0,C 180,E1 -9047.799,E2 -9047.799} C_VEL
LIN {X 0,Y 439.393,Z 214.754,A -85,B 0,C 180,E1 -9050.229,E2 -9050.229} C_VEL
LIN {X 0,Y 439.359,Z 214.757,A -85,B 0,C 180,E1 -9053.716,E2 -9053.716} C_VEL
LIN {X 0,Y 439.36,Z 214.755,A -85,B 0,C 180,E1 -9057.057,E2 -9057.057} C_VEL
LIN {X 0,Y 439.372,Z 214.758,A -85,B 0,C 180,E1 -9060.277,E2 -9060.277} C_VEL
LIN {X 0,Y 439.477,Z 214.817,A -85,B 0,C 180,E1 -9062.825,E2 -9062.825} C_VEL
LIN {X 0,Y 441.751,Z 226.392,A -85,B 0,C 180,E1 -9065.073,E2 -9065.073} C_VEL
LIN {X 0,Y 442.04,Z 230.538,A -85,B 0,C 180,E1 -9065.836,E2 -9065.836} C_VEL
LIN {X 0,Y 441.151,Z 247.138,A -85,B 0,C 180,E1 -9068.753,E2 -9068.753} C_VEL
LIN {X 0,Y 440.458,Z 264.317,A -85,B 0,C 180,E1 -9071.726,E2 -9071.726} C_VEL
LIN {X 0,Y 444.143,Z 289.329,A -85,B 0,C 180,E1 -9072.348,E2 -9072.348} C_VEL
LIN {X 0,Y 443.129,Z 374.478,A -85,B 0,C 180,E1 -9073.858,E2 -9073.858} C_VEL
LIN {X 0,Y 442.624,Z 387.168,A -85,B 0,C 180,E1 -9074.253,E2 -9074.253} C_VEL
LIN {X 0,Y 441.994,Z 400.21,A -85,B 0,C 180,E1 -9074.85,E2 -9074.85} C_VEL
LIN {X 0,Y 441.382,Z 412.082,A -85,B 0,C 180,E1 -9075.596,E2 -9075.596} C_VEL
LIN {X 0,Y 440.771,Z 423.342,A -85,B 0,C 180,E1 -9076.498,E2 -9076.498} C_VEL
LIN {X 0,Y 440.116,Z 433.912,A -85,B 0,C 180,E1 -9077.552,E2 -9077.552} C_VEL
LIN {X 0,Y 439.607,Z 443.237,A -85,B 0,C 180,E1 -9078.707,E2 -9078.707} C_VEL
LIN {X 0,Y 439.072,Z 452.323,A -85,B 0,C 180,E1 -9080.093,E2 -9080.093} C_VEL
LIN {X 0,Y 438.7,Z 459.653,A -85,B 0,C 180,E1 -9081.479,E2 -9081.479} C_VEL
LIN {X 0,Y 438.523,Z 464.608,A -85,B 0,C 180,E1 -9082.634,E2 -9082.634} C_VEL
LIN {X 0,Y 438.344,Z 469.455,A -85,B 0,C 180,E1 -9084.028,E2 -9084.028} C_VEL
LIN {X 0,Y 438.345,Z 473.114,A -85,B 0,C 180,E1 -9085.402,E2 -9085.402} C_VEL
LIN {X 0,Y 438.293,Z 475.01,A -85,B 0,C 180,E1 -9086.323,E2 -9086.323} C_VEL
LIN {X 0,Y 438.373,Z 476.439,A -85,B 0,C 180,E1 -9087.243,E2 -9087.243} C_VEL
LIN {X 0,Y 438.309,Z 478.084,A -85,B 0,C 180,E1 -9089.081,E2 -9089.081} C_VEL
LIN {X 0,Y 438.315,Z 478.291,A -85,B 0,C 180,E1 -9090,E2 -9090} C_VEL
LIN {X 0,Y 438.308,Z 478.063,A -85,B 0,C 180,E1 -9090.919,E2 -9090.919} C_VEL
LIN {X 0,Y 438.371,Z 476.42,A -85,B 0,C 180,E1 -9092.756,E2 -9092.756} C_VEL
LIN {X 0,Y 438.29,Z 474.956,A -85,B 0,C 180,E1 -9093.677,E2 -9093.677} C_VEL
LIN {X 0,Y 438.407,Z 471.938,A -85,B 0,C 180,E1 -9095.058,E2 -9095.058} C_VEL
LIN {X 0,Y 438.448,Z 467.836,A -85,B 0,C 180,E1 -9096.442,E2 -9096.442} C_VEL
LIN {X 0,Y 438.654,Z 461.524,A -85,B 0,C 180,E1 -9098.058,E2 -9098.058} C_VEL
LIN {X 0,Y 438.931,Z 454.641,A -85,B 0,C 180,E1 -9099.445,E2 -9099.445} C_VEL
LIN {X 0,Y 439.35,Z 446.054,A -85,B 0,C 180,E1 -9100.832,E2 -9100.832} C_VEL
LIN {X 0,Y 439.87,Z 437.219,A -85,B 0,C 180,E1 -9101.987,E2 -9101.987} C_VEL
LIN {X 0,Y 440.513,Z 426.435,A -85,B 0,C 180,E1 -9103.131,E2 -9103.131} C_VEL
LIN {X 0,Y 441.084,Z 415.459,A -85,B 0,C 180,E1 -9104.061,E2 -9104.061} C_VEL
LIN {X 0,Y 441.648,Z 403.254,A -85,B 0,C 180,E1 -9104.867,E2 -9104.867} C_VEL
LIN {X 0,Y 442.235,Z 390.542,A -85,B 0,C 180,E1 -9105.495,E2 -9105.495} C_VEL
LIN {X 0,Y 442.705,Z 378.016,A -85,B 0,C 180,E1 -9105.921,E2 -9105.921} C_VEL
LIN {X 0,Y 443.024,Z 360.772,A -85,B 0,C 180,E1 -9106.264,E2 -9106.264} C_VEL
LIN {X 0,Y 443.63,Z 288.016,A -85,B 0,C 180,E1 -9107.515,E2 -9107.515} C_VEL
LIN {X 0,Y 440.337,Z 265.539,A -85,B 0,C 180,E1 -9108.056,E2 -9108.056} C_VEL
LIN {X 0,Y 441.159,Z 249.069,A -85,B 0,C 180,E1 -9111.002,E2 -9111.002} C_VEL
LIN {X 0,Y 442.187,Z 231.631,A -85,B 0,C 180,E1 -9114.156,E2 -9114.156} C_VEL
LIN {X 0,Y 441.837,Z 226.404,A -85,B 0,C 180,E1 -9115.144,E2 -9115.144} C_VEL
LIN {X 0,Y 439.49,Z 214.742,A -85,B 0,C 180,E1 -9117.496,E2 -9117.496} C_VEL
LIN {X 0,Y 439.349,Z 214.757,A -85,B 0,C 180,E1 -9120.786,E2 -9120.786} C_VEL
LIN {X 0,Y 439.374,Z 214.758,A -85,B 0,C 180,E1 -9124.04,E2 -9124.04} C_VEL
LIN {X 0,Y 439.332,Z 214.756,A -85,B 0,C 180,E1 -9126.884,E2 -9126.884} C_VEL
LIN {X 0,Y 439.383,Z 214.756,A -85,B 0,C 180,E1 -9129.846,E2 -9129.846} C_VEL
LIN {X 0,Y 439.359,Z 214.753,A -85,B 0,C 180,E1 -9132.623,E2 -9132.623} C_VEL
LIN {X 0,Y 439.376,Z 214.752,A -85,B 0,C 180,E1 -9135.267,E2 -9135.267} C_VEL
LIN {X 0,Y 439.36,Z 214.752,A -85,B 0,C 180,E1 -9138.74,E2 -9138.74} C_VEL
LIN {X 0,Y 439.339,Z 214.762,A -85,B 0,C 180,E1 -9141.605,E2 -9141.605} C_VEL
LIN {X 0,Y 439.367,Z 214.752,A -85,B 0,C 180,E1 -9144.841,E2 -9144.841} C_VEL
LIN {X 0,Y 439.336,Z 214.756,A -85,B 0,C 180,E1 -9148.136,E2 -9148.136} C_VEL
LIN {X 0,Y 439.395,Z 214.754,A -85,B 0,C 180,E1 -9151.595,E2 -9151.595} C_VEL
LIN {X 0,Y 439.364,Z 214.751,A -85,B 0,C 180,E1 -9154.412,E2 -9154.412} C_VEL
LIN {X 0,Y 439.324,Z 214.764,A -85,B 0,C 180,E1 -9157.422,E2 -9157.422} C_VEL
LIN {X 0,Y 439.397,Z 214.748,A -85,B 0,C 180,E1 -9160.661,E2 -9160.661} C_VEL
LIN {X 0,Y 439.416,Z 214.745,A -85,B 0,C 180,E1 -9164.222,E2 -9164.222} C_VEL
LIN {X 0,Y 439.46,Z 214.74,A -85,B 0,C 180,E1 -9168,E2 -9168} C_VEL
LIN {X 0,Y 439.5,Z 214.736,A -85,B 0,C 180,E1 -9171.725,E2 -9171.725} C_VEL
LIN {X 0,Y 439.564,Z 214.728,A -85,B 0,C 180,E1 -9174.495,E2 -9174.495} C_VEL
LIN {X 0,Y 439.582,Z 214.725,A -85,B 0,C 180,E1 -9178.167,E2 -9178.167} C_VEL
LIN {X 0,Y 439.709,Z 214.709,A -85,B 0,C 180,E1 -9180,E2 -9180} C_VEL
LIN {X 0,Y 439.59,Z 214.729,A -85,B 0,C 180,E1 -9182.749,E2 -9182.749} C_VEL
LIN {X 0,Y 439.581,Z 214.728,A -85,B 0,C 180,E1 -9186.425,E2 -9186.425} C_VEL
LIN {X 0,Y 439.453,Z 214.743,A -85,B 0,C 180,E1 -9189.202,E2 -9189.202} C_VEL
LIN {X 0,Y 439.457,Z 214.747,A -85,B 0,C 180,E1 -9192.728,E2 -9192.728} C_VEL
LIN {X 0,Y 439.414,Z 214.75,A -85,B 0,C 180,E1 -9196.355,E2 -9196.355} C_VEL
LIN {X 0,Y 439.397,Z 214.748,A -85,B 0,C 180,E1 -9199.626,E2 -9199.626} C_VEL
LIN {X 0,Y 439.388,Z 214.755,A -85,B 0,C 180,E1 -9202.574,E2 -9202.574} C_VEL
LIN {X 0,Y 439.372,Z 214.751,A -85,B 0,C 180,E1 -9205.587,E2 -9205.587} C_VEL
LIN {X 0,Y 439.386,Z 214.753,A -85,B 0,C 180,E1 -9208.675,E2 -9208.675} C_VEL
LIN {X 0,Y 439.335,Z 214.758,A -85,B 0,C 180,E1 -9211.863,E2 -9211.863} C_VEL
LIN {X 0,Y 439.364,Z 214.752,A -85,B 0,C 180,E1 -9215.159,E2 -9215.159} C_VEL
LIN {X 0,Y 439.368,Z 214.754,A -85,B 0,C 180,E1 -9218.596,E2 -9218.596} C_VEL
LIN {X 0,Y 439.373,Z 214.751,A -85,B 0,C 180,E1 -9221.262,E2 -9221.262} C_VEL
LIN {X 0,Y 439.381,Z 214.75,A -85,B 0,C 180,E1 -9224.731,E2 -9224.731} C_VEL
LIN {X 0,Y 439.372,Z 214.755,A -85,B 0,C 180,E1 -9227.799,E2 -9227.799} C_VEL
LIN {X 0,Y 439.426,Z 214.748,A -85,B 0,C 180,E1 -9230.233,E2 -9230.233} C_VEL
LIN {X 0,Y 439.357,Z 214.758,A -85,B 0,C 180,E1 -9233.716,E2 -9233.716} C_VEL
LIN {X 0,Y 439.356,Z 214.753,A -85,B 0,C 180,E1 -9237.057,E2 -9237.057} C_VEL
LIN {X 0,Y 439.382,Z 214.751,A -85,B 0,C 180,E1 -9240.278,E2 -9240.278} C_VEL
LIN {X 0,Y 439.419,Z 214.749,A -85,B 0,C 180,E1 -9243.399,E2 -9243.399} C_VEL
LIN {X 0,Y 439.377,Z 214.75,A -85,B 0,C 180,E1 -9246.432,E2 -9246.432} C_VEL
LIN {X 0,Y 439.38,Z 214.755,A -85,B 0,C 180,E1 -9249.399,E2 -9249.399} C_VEL
LIN {X 0,Y 439.425,Z 214.744,A -85,B 0,C 180,E1 -9252.311,E2 -9252.311} C_VEL
LIN {X 0,Y 439.444,Z 214.745,A -85,B 0,C 180,E1 -9255.176,E2 -9255.176} C_VEL
LIN {X 0,Y 439.48,Z 214.739,A -85,B 0,C 180,E1 -9258.003,E2 -9258.003} C_VEL
LIN {X 0,Y 439.546,Z 214.732,A -85,B 0,C 180,E1 -9261.727,E2 -9261.727} C_VEL
LIN {X 0,Y 439.616,Z 214.72,A -85,B 0,C 180,E1 -9264.496,E2 -9264.496} C_VEL
LIN {X 0,Y 439.633,Z 214.718,A -85,B 0,C 180,E1 -9268.168,E2 -9268.168} C_VEL
LIN {X 0,Y 439.761,Z 214.702,A -85,B 0,C 180,E1 -9270,E2 -9270} C_VEL
LIN {X 0,Y 439.607,Z 214.724,A -85,B 0,C 180,E1 -9271.036,E2 -9271.036} C_VEL
LIN {X 0,Y 438.904,Z 214.811,A -85,B 0,C 180,E1 -9271.8,E2 -9271.8} C_VEL
LIN {X 0,Y 435.932,Z 215.185,A -85,B 0,C 180,E1 -9273.04,E2 -9273.04} C_VEL
LIN {X 0,Y 433.48,Z 215.489,A -85,B 0,C 180,E1 -9274.04,E2 -9274.04} C_VEL
LIN {X 0,Y 432.506,Z 215.61,A -85,B 0,C 180,E1 -9274.815,E2 -9274.815} C_VEL
LIN {X 0,Y 432.468,Z 215.611,A -85,B 0,C 180,E1 -9275.077,E2 -9275.077} C_VEL
LIN {X 0,Y 432.536,Z 215.604,A -85,B 0,C 180,E1 -9277.632,E2 -9277.632} C_VEL
LIN {X 0,Y 432.39,Z 215.625,A -85,B 0,C 180,E1 -9281.246,E2 -9281.246} C_VEL
LIN {X 0,Y 432.369,Z 215.623,A -85,B 0,C 180,E1 -9284.111,E2 -9284.111} C_VEL
LIN {X 0,Y 432.392,Z 215.626,A -85,B 0,C 180,E1 -9287.01,E2 -9287.01} C_VEL
LIN {X 0,Y 432.332,Z 215.628,A -85,B 0,C 180,E1 -9289.959,E2 -9289.959} C_VEL
LIN {X 0,Y 432.31,Z 215.635,A -85,B 0,C 180,E1 -9292.962,E2 -9292.962} C_VEL
LIN {X 0,Y 432.354,Z 215.629,A -85,B 0,C 180,E1 -9296.03,E2 -9296.03} C_VEL
LIN {X 0,Y 432.43,Z 215.723,A -85,B 0,C 180,E1 -9299.098,E2 -9299.098} C_VEL
LIN {X 0,Y 433.784,Z 223.138,A -85,B 0,C 180,E1 -9300.831,E2 -9300.831} C_VEL
LIN {X 0,Y 433.722,Z 227.424,A -85,B 0,C 180,E1 -9301.774,E2 -9301.774} C_VEL
LIN {X 0,Y 437.24,Z 245.794,A -85,B 0,C 180,E1 -9302.252,E2 -9302.252} C_VEL
LIN {X 0,Y 436.096,Z 334.973,A -85,B 0,C 180,E1 -9303.827,E2 -9303.827} C_VEL
LIN {X 0,Y 435.699,Z 348.22,A -85,B 0,C 180,E1 -9304.245,E2 -9304.245} C_VEL
LIN {X 0,Y 435.36,Z 360.986,A -85,B 0,C 180,E1 -9304.846,E2 -9304.846} C_VEL
LIN {X 0,Y 434.83,Z 372.509,A -85,B 0,C 180,E1 -9305.577,E2 -9305.577} C_VEL
LIN {X 0,Y 434.237,Z 383.663,A -85,B 0,C 180,E1 -9306.48,E2 -9306.48} C_VEL
LIN {X 0,Y 433.676,Z 393.924,A -85,B 0,C 180,E1 -9307.515,E2 -9307.515} C_VEL
LIN {X 0,Y 433.142,Z 402.951,A -85,B 0,C 180,E1 -9308.633,E2 -9308.633} C_VEL
LIN {X 0,Y 432.64,Z 411.729,A -85,B 0,C 180,E1 -9309.978,E2 -9309.978} C_VEL
LIN {X 0,Y 432.139,Z 418.809,A -85,B 0,C 180,E1 -9311.31,E2 -9311.31} C_VEL
LIN {X 0,Y 431.821,Z 425.576,A -85,B 0,C 180,E1 -9312.914,E2 -9312.914} C_VEL
LIN {X 0,Y 431.563,Z 430.483,A -85,B 0,C 180,E1 -9314.441,E2 -9314.441} C_VEL
LIN {X 0,Y 431.388,Z 433.763,A -85,B 0,C 180,E1 -9315.787,E2 -9315.787} C_VEL
LIN {X 0,Y 431.251,Z 436.16,A -85,B 0,C 180,E1 -9317.162,E2 -9317.162} C_VEL
LIN {X 0,Y 431.17,Z 437.661,A -85,B 0,C 180,E1 -9318.565,E2 -9318.565} C_VEL
LIN {X 0,Y 431.113,Z 438.25,A -85,B 0,C 180,E1 -9320.006,E2 -9320.006} C_VEL
LIN {X 0,Y 431.127,Z 437.709,A -85,B 0,C 180,E1 -9321.724,E2 -9321.724} C_VEL
LIN {X 0,Y 431.227,Z 436.437,A -85,B 0,C 180,E1 -9322.987,E2 -9322.987} C_VEL
LIN {X 0,Y 431.39,Z 433.846,A -85,B 0,C 180,E1 -9324.537,E2 -9324.537} C_VEL
LIN {X 0,Y 431.606,Z 429.87,A -85,B 0,C 180,E1 -9326.136,E2 -9326.136} C_VEL
LIN {X 0,Y 432.005,Z 424.338,A -85,B 0,C 180,E1 -9327.764,E2 -9327.764} C_VEL
LIN {X 0,Y 432.363,Z 418.6,A -85,B 0,C 180,E1 -9329.088,E2 -9329.088} C_VEL
LIN {X 0,Y 432.944,Z 410.472,A -85,B 0,C 180,E1 -9330.591,E2 -9330.591} C_VEL
LIN {X 0,Y 433.591,Z 401.094,A -85,B 0,C 180,E1 -9331.962,E2 -9331.962} C_VEL
LIN {X 0,Y 434.179,Z 390.784,A -85,B 0,C 180,E1 -9333.179,E2 -9333.179} C_VEL
LIN {X 0,Y 434.881,Z 379.677,A -85,B 0,C 180,E1 -9334.212,E2 -9334.212} C_VEL
LIN {X 0,Y 435.485,Z 368.559,A -85,B 0,C 180,E1 -9335.034,E2 -9335.034} C_VEL
LIN {X 0,Y 436.043,Z 356.26,A -85,B 0,C 180,E1 -9335.733,E2 -9335.733} C_VEL
LIN {X 0,Y 436.44,Z 343.145,A -85,B 0,C 180,E1 -9336.261,E2 -9336.261} C_VEL
LIN {X 0,Y 436.719,Z 329.954,A -85,B 0,C 180,E1 -9336.598,E2 -9336.598} C_VEL
LIN {X 0,Y 437.82,Z 244.707,A -85,B 0,C 180,E1 -9338.117,E2 -9338.117} C_VEL
LIN {X 0,Y 434.137,Z 227.711,A -85,B 0,C 180,E1 -9338.64,E2 -9338.64} C_VEL
LIN {X 0,Y 433.908,Z 222.832,A -85,B 0,C 180,E1 -9339.621,E2 -9339.621} C_VEL
LIN {X 0,Y 432.383,Z 215.627,A -85,B 0,C 180,E1 -9341.153,E2 -9341.153} C_VEL
LIN {X 0,Y 432.397,Z 215.626,A -85,B 0,C 180,E1 -9343.96,E2 -9343.96} C_VEL
LIN {X 0,Y 432.438,Z 215.624,A -85,B 0,C 180,E1 -9347.803,E2 -9347.803} C_VEL
LIN {X 0,Y 432.445,Z 215.62,A -85,B 0,C 180,E1 -9351.59,E2 -9351.59} C_VEL
LIN {X 0,Y 432.557,Z 215.603,A -85,B 0,C 180,E1 -9354.406,E2 -9354.406} C_VEL
LIN {X 0,Y 432.553,Z 215.602,A -85,B 0,C 180,E1 -9358.138,E2 -9358.138} C_VEL
LIN {X 0,Y 432.681,Z 215.587,A -85,B 0,C 180,E1 -9360,E2 -9360} C_VEL
LIN {X 0,Y 432.542,Z 215.608,A -85,B 0,C 180,E1 -9362.794,E2 -9362.794} C_VEL
LIN {X 0,Y 432.518,Z 215.606,A -85,B 0,C 180,E1 -9366.531,E2 -9366.531} C_VEL
LIN {X 0,Y 432.398,Z 215.623,A -85,B 0,C 180,E1 -9369.354,E2 -9369.354} C_VEL
LIN {X 0,Y 432.4,Z 215.626,A -85,B 0,C 180,E1 -9372.812,E2 -9372.812} C_VEL
LIN {X 0,Y 432.379,Z 215.627,A -85,B 0,C 180,E1 -9376.485,E2 -9376.485} C_VEL
LIN {X 0,Y 432.296,Z 215.633,A -85,B 0,C 180,E1 -9379.963,E2 -9379.963} C_VEL
LIN {X 0,Y 432.279,Z 215.635,A -85,B 0,C 180,E1 -9382.967,E2 -9382.967} C_VEL
LIN {X 0,Y 432.326,Z 215.631,A -85,B 0,C 180,E1 -9386.035,E2 -9386.035} C_VEL
LIN {X 0,Y 432.306,Z 215.63,A -85,B 0,C 180,E1 -9389.191,E2 -9389.191} C_VEL
LIN {X 0,Y 432.289,Z 215.636,A -85,B 0,C 180,E1 -9392.446,E2 -9392.446} C_VEL
LIN {X 0,Y 432.314,Z 215.628,A -85,B 0,C 180,E1 -9395.635,E2 -9395.635} C_VEL
LIN {X 0,Y 432.304,Z 215.636,A -85,B 0,C 180,E1 -9398.716,E2 -9398.716} C_VEL
LIN {X 0,Y 432.304,Z 215.634,A -85,B 0,C 180,E1 -9401.801,E2 -9401.801} C_VEL
LIN {X 0,Y 432.311,Z 215.636,A -85,B 0,C 180,E1 -9404.351,E2 -9404.351} C_VEL
LIN {X 0,Y 432.298,Z 215.633,A -85,B 0,C 180,E1 -9407.019,E2 -9407.019} C_VEL
LIN {X 0,Y 432.315,Z 215.634,A -85,B 0,C 180,E1 -9409.824,E2 -9409.824} C_VEL
LIN {X 0,Y 432.291,Z 215.635,A -85,B 0,C 180,E1 -9413.025,E2 -9413.025} C_VEL
LIN {X 0,Y 432.347,Z 215.633,A -85,B 0,C 180,E1 -9416,E2 -9416} C_VEL
LIN {X 0,Y 432.337,Z 215.633,A -85,B 0,C 180,E1 -9419.493,E2 -9419.493} C_VEL
LIN {X 0,Y 432.434,Z 215.683,A -85,B 0,C 180,E1 -9422.542,E2 -9422.542} C_VEL
LIN {X 0,Y 434.772,Z 227.326,A -85,B 0,C 180,E1 -9424.855,E2 -9424.855} C_VEL
LIN {X 0,Y 435.139,Z 231.721,A -85,B 0,C 180,E1 -9425.681,E2 -9425.681} C_VEL
LIN {X 0,Y 434.301,Z 246.951,A -85,B 0,C 180,E1 -9428.401,E2 -9428.401} C_VEL
LIN {X 0,Y 433.493,Z 263.811,A -85,B 0,C 180,E1 -9431.388,E2 -9431.388} C_VEL
LIN {X 0,Y 436.967,Z 286.605,A -85,B 0,C 180,E1 -9431.979,E2 -9431.979} C_VEL
LIN {X 0,Y 437.363,Z 291.484,A -85,B 0,C 180,E1 -9432.088,E2 -9432.088} C_VEL
LIN {X 0,Y 436.363,Z 373.718,A -85,B 0,C 180,E1 -9433.571,E2 -9433.571} C_VEL
LIN {X 0,Y 435.803,Z 387.279,A -85,B 0,C 180,E1 -9434,E2 -9434} C_VEL
LIN {X 0,Y 435.159,Z 400.149,A -85,B 0,C 180,E1 -9434.607,E2 -9434.607} C_VEL
LIN {X 0,Y 434.505,Z 411.939,A -85,B 0,C 180,E1 -9435.362,E2 -9435.362} C_VEL
LIN {X 0,Y 433.816,Z 423.645,A -85,B 0,C 180,E1 -9436.323,E2 -9436.323} C_VEL
LIN {X 0,Y 433.146,Z 433.674,A -85,B 0,C 180,E1 -9437.348,E2 -9437.348} C_VEL
LIN {X 0,Y 432.616,Z 442.976,A -85,B 0,C 180,E1 -9438.522,E2 -9438.522} C_VEL
LIN {X 0,Y 432.01,Z 452.054,A -85,B 0,C 180,E1 -9439.929,E2 -9439.929} C_VEL
LIN {X 0,Y 431.653,Z 459.372,A -85,B 0,C 180,E1 -9441.339,E2 -9441.339} C_VEL
LIN {X 0,Y 431.438,Z 464.318,A -85,B 0,C 180,E1 -9442.513,E2 -9442.513} C_VEL
LIN {X 0,Y 431.245,Z 469.584,A -85,B 0,C 180,E1 -9444.07,E2 -9444.07} C_VEL
LIN {X 0,Y 431.272,Z 472.809,A -85,B 0,C 180,E1 -9445.327,E2 -9445.327} C_VEL
LIN {X 0,Y 431.199,Z 474.698,A -85,B 0,C 180,E1 -9446.262,E2 -9446.262} C_VEL
LIN {X 0,Y 431.281,Z 476.124,A -85,B 0,C 180,E1 -9447.198,E2 -9447.198} C_VEL
LIN {X 0,Y 431.241,Z 477.141,A -85,B 0,C 180,E1 -9448.132,E2 -9448.132} C_VEL
LIN {X 0,Y 431.222,Z 477.762,A -85,B 0,C 180,E1 -9449.066,E2 -9449.066} C_VEL
LIN {X 0,Y 431.226,Z 477.96,A -85,B 0,C 180,E1 -9450,E2 -9450} C_VEL
LIN {X 0,Y 431.222,Z 477.726,A -85,B 0,C 180,E1 -9450.934,E2 -9450.934} C_VEL
LIN {X 0,Y 431.241,Z 477.098,A -85,B 0,C 180,E1 -9451.868,E2 -9451.868} C_VEL
LIN {X 0,Y 431.279,Z 476.071,A -85,B 0,C 180,E1 -9452.802,E2 -9452.802} C_VEL
LIN {X 0,Y 431.196,Z 474.593,A -85,B 0,C 180,E1 -9453.738,E2 -9453.738} C_VEL
LIN {X 0,Y 431.312,Z 471.559,A -85,B 0,C 180,E1 -9455.141,E2 -9455.141} C_VEL
LIN {X 0,Y 431.376,Z 467.439,A -85,B 0,C 180,E1 -9456.548,E2 -9456.548} C_VEL
LIN {X 0,Y 431.585,Z 461.103,A -85,B 0,C 180,E1 -9458.191,E2 -9458.191} C_VEL
LIN {X 0,Y 431.878,Z 454.194,A -85,B 0,C 180,E1 -9459.601,E2 -9459.601} C_VEL
LIN {X 0,Y 432.232,Z 447.139,A -85,B 0,C 180,E1 -9460.776,E2 -9460.776} C_VEL
LIN {X 0,Y 432.784,Z 438.645,A -85,B 0,C 180,E1 -9461.948,E2 -9461.948} C_VEL
LIN {X 0,Y 433.399,Z 428.141,A -85,B 0,C 180,E1 -9463.12,E2 -9463.12} C_VEL
LIN {X 0,Y 434.069,Z 416.316,A -85,B 0,C 180,E1 -9464.174,E2 -9464.174} C_VEL
LIN {X 0,Y 434.672,Z 404.485,A -85,B 0,C 180,E1 -9464.991,E2 -9464.991} C_VEL
LIN {X 0,Y 435.316,Z 390.942,A -85,B 0,C 180,E1 -9465.687,E2 -9465.687} C_VEL
LIN {X 0,Y 435.832,Z 377.823,A -85,B 0,C 180,E1 -9466.149,E2 -9466.149} C_VEL
LIN {X 0,Y 436.165,Z 360.709,A -85,B 0,C 180,E1 -9466.497,E2 -9466.497} C_VEL
LIN {X 0,Y 436.79,Z 288.563,A -85,B 0,C 180,E1 -9467.762,E2 -9467.762} C_VEL
LIN {X 0,Y 433.397,Z 265.309,A -85,B 0,C 180,E1 -9468.321,E2 -9468.321} C_VEL
LIN {X 0,Y 434.353,Z 247.307,A -85,B 0,C 180,E1 -9471.596,E2 -9471.596} C_VEL
LIN {X 0,Y 435.294,Z 231.221,A -85,B 0,C 180,E1 -9474.563,E2 -9474.563} C_VEL
LIN {X 0,Y 434.407,Z 225.483,A -85,B 0,C 180,E1 -9475.693,E2 -9475.693} C_VEL
LIN {X 0,Y 432.44,Z 215.62,A -85,B 0,C 180,E1 -9477.721,E2 -9477.721} C_VEL
LIN {X 0,Y 432.309,Z 215.634,A -85,B 0,C 180,E1 -9481.343,E2 -9481.343} C_VEL
LIN {X 0,Y 432.326,Z 215.629,A -85,B 0,C 180,E1 -9484.674,E2 -9484.674} C_VEL
LIN {X 0,Y 432.319,Z 215.634,A -85,B 0,C 180,E1 -9488.147,E2 -9488.147} C_VEL
LIN {X 0,Y 432.312,Z 215.634,A -85,B 0,C 180,E1 -9491.598,E2 -9491.598} C_VEL
LIN {X 0,Y 432.311,Z 215.632,A -85,B 0,C 180,E1 -9494.344,E2 -9494.344} C_VEL
LIN {X 0,Y 432.295,Z 215.633,A -85,B 0,C 180,E1 -9497.012,E2 -9497.012} C_VEL
LIN {X 0,Y 432.306,Z 215.637,A -85,B 0,C 180,E1 -9499.817,E2 -9499.817} C_VEL
LIN {X 0,Y 432.275,Z 215.636,A -85,B 0,C 180,E1 -9503.018,E2 -9503.018} C_VEL
LIN {X 0,Y 432.327,Z 215.631,A -85,B 0,C 180,E1 -9505.993,E2 -9505.993} C_VEL
LIN {X 0,Y 432.31,Z 215.638,A -85,B 0,C 180,E1 -9509.487,E2 -9509.487} C_VEL
LIN {X 0,Y 432.352,Z 215.627,A -85,B 0,C 180,E1 -9512.925,E2 -9512.925} C_VEL
LIN {X 0,Y 432.33,Z 215.629,A -85,B 0,C 180,E1 -9516.021,E2 -9516.021} C_VEL
LIN {X 0,Y 432.307,Z 215.635,A -85,B 0,C 180,E1 -9519.044,E2 -9519.044} C_VEL
LIN {X 0,Y 432.333,Z 215.628,A -85,B 0,C 180,E1 -9522.009,E2 -9522.009} C_VEL
LIN {X 0,Y 432.347,Z 215.63,A -85,B 0,C 180,E1 -9524.924,E2 -9524.924} C_VEL
LIN {X 0,Y 432.434,Z 215.616,A -85,B 0,C 180,E1 -9527.802,E2 -9527.802} C_VEL
LIN {X 0,Y 432.444,Z 215.616,A -85,B 0,C 180,E1 -9531.589,E2 -9531.589} C_VEL
LIN {X 0,Y 432.541,Z 215.603,A -85,B 0,C 180,E1 -9534.405,E2 -9534.405} C_VEL
LIN {X 0,Y 432.552,Z 215.6,A -85,B 0,C 180,E1 -9538.137,E2 -9538.137} C_VEL
LIN {X 0,Y 432.679,Z 215.584,A -85,B 0,C 180,E1 -9540,E2 -9540} C_VEL
LIN {X 0,Y 432.543,Z 215.608,A -85,B 0,C 180,E1 -9542.794,E2 -9542.794} C_VEL
LIN {X 0,Y 432.555,Z 215.604,A -85,B 0,C 180,E1 -9546.53,E2 -9546.53} C_VEL
LIN {X 0,Y 432.397,Z 215.621,A -85,B 0,C 180,E1 -9549.354,E2 -9549.354} C_VEL
LIN {X 0,Y 432.399,Z 215.625,A -85,B 0,C 180,E1 -9552.813,E2 -9552.813} C_VEL
LIN {X 0,Y 432.377,Z 215.628,A -85,B 0,C 180,E1 -9556.484,E2 -9556.484} C_VEL
LIN {X 0,Y 432.346,Z 215.627,A -85,B 0,C 180,E1 -9559.96,E2 -9559.96} C_VEL
LIN {X 0,Y 432.319,Z 215.631,A -85,B 0,C 180,E1 -9562.964,E2 -9562.964} C_VEL
LIN {X 0,Y 432.327,Z 215.631,A -85,B 0,C 180,E1 -9566.034,E2 -9566.034} C_VEL
LIN {X 0,Y 432.313,Z 215.63,A -85,B 0,C 180,E1 -9569.189,E2 -9569.189} C_VEL
LIN {X 0,Y 432.288,Z 215.641,A -85,B 0,C 180,E1 -9572.296,E2 -9572.296} C_VEL
LIN {X 0,Y 432.305,Z 215.634,A -85,B 0,C 180,E1 -9574.68,E2 -9574.68} C_VEL
LIN {X 0,Y 432.321,Z 215.636,A -85,B 0,C 180,E1 -9578.151,E2 -9578.151} C_VEL
LIN {X 0,Y 432.342,Z 215.628,A -85,B 0,C 180,E1 -9581.611,E2 -9581.611} C_VEL
LIN {X 0,Y 432.335,Z 215.631,A -85,B 0,C 180,E1 -9584.347,E2 -9584.347} C_VEL
LIN {X 0,Y 432.341,Z 215.631,A -85,B 0,C 180,E1 -9588.21,E2 -9588.21} C_VEL
LIN {X 0,Y 432.336,Z 215.628,A -85,B 0,C 180,E1 -9591.286,E2 -9591.286} C_VEL
LIN {X 0,Y 432.326,Z 215.63,A -85,B 0,C 180,E1 -9594.371,E2 -9594.371} C_VEL
LIN {X 0,Y 432.307,Z 215.635,A -85,B 0,C 180,E1 -9597.56,E2 -9597.56} C_VEL
LIN {X 0,Y 432.38,Z 215.629,A -85,B 0,C 180,E1 -9599.747,E2 -9599.747} C_VEL
LIN {X 0,Y 432.389,Z 215.624,A -85,B 0,C 180,E1 -9603.375,E2 -9603.375} C_VEL
LIN {X 0,Y 432.362,Z 215.627,A -85,B 0,C 180,E1 -9606.026,E2 -9606.026} C_VEL
LIN {X 0,Y 432.342,Z 215.628,A -85,B 0,C 180,E1 -9609.048,E2 -9609.048} C_VEL
LIN {X 0,Y 432.372,Z 215.625,A -85,B 0,C 180,E1 -9612.013,E2 -9612.013} C_VEL
LIN {X 0,Y 432.391,Z 215.622,A -85,B 0,C 180,E1 -9614.928,E2 -9614.928} C_VEL
LIN {X 0,Y 432.455,Z 215.615,A -85,B 0,C 180,E1 -9617.805,E2 -9617.805} C_VEL
LIN {X 0,Y 432.49,Z 215.613,A -85,B 0,C 180,E1 -9621.591,E2 -9621.591} C_VEL
LIN {X 0,Y 432.592,Z 215.595,A -85,B 0,C 180,E1 -9624.407,E2 -9624.407} C_VEL
LIN {X 0,Y 432.603,Z 215.594,A -85,B 0,C 180,E1 -9628.138,E2 -9628.138} C_VEL
LIN {X 0,Y 432.731,Z 215.578,A -85,B 0,C 180,E1 -9630,E2 -9630} C_VEL
LIN {X 0,Y 432.604,Z 215.597,A -85,B 0,C 180,E1 -9632.793,E2 -9632.793} C_VEL
LIN {X 0,Y 432.468,Z 215.611,A -85,B 0,C 180,E1 -9635.077,E2 -9635.077} C_VEL
LIN {X 0,Y 431.906,Z 215.683,A -85,B 0,C 180,E1 -9635.855,E2 -9635.855} C_VEL
LIN {X 0,Y 429.052,Z 216.043,A -85,B 0,C 180,E1 -9637.119,E2 -9637.119} C_VEL
LIN {X 0,Y 426.564,Z 216.349,A -85,B 0,C 180,E1 -9638.139,E2 -9638.139} C_VEL
LIN {X 0,Y 425.486,Z 216.487,A -85,B 0,C 180,E1 -9638.929,E2 -9638.929} C_VEL
LIN {X 0,Y 425.397,Z 216.492,A -85,B 0,C 180,E1 -9639.196,E2 -9639.196} C_VEL
LIN {X 0,Y 425.39,Z 216.499,A -85,B 0,C 180,E1 -9642.902,E2 -9642.902} C_VEL
LIN {X 0,Y 425.356,Z 216.501,A -85,B 0,C 180,E1 -9646.603,E2 -9646.603} C_VEL
LIN {X 0,Y 425.322,Z 216.501,A -85,B 0,C 180,E1 -9649.634,E2 -9649.634} C_VEL
LIN {X 0,Y 425.279,Z 216.509,A -85,B 0,C 180,E1 -9652.337,E2 -9652.337} C_VEL
LIN {X 0,Y 425.285,Z 216.509,A -85,B 0,C 180,E1 -9655.443,E2 -9655.443} C_VEL
LIN {X 0,Y 425.361,Z 216.503,A -85,B 0,C 180,E1 -9658.627,E2 -9658.627} C_VEL
LIN {X 0,Y 425.407,Z 216.75,A -85,B 0,C 180,E1 -9658.941,E2 -9658.941} C_VEL
LIN {X 0,Y 426.804,Z 224.109,A -85,B 0,C 180,E1 -9660.691,E2 -9660.691} C_VEL
LIN {X 0,Y 426.805,Z 227.789,A -85,B 0,C 180,E1 -9661.496,E2 -9661.496} C_VEL
LIN {X 0,Y 430.426,Z 245.726,A -85,B 0,C 180,E1 -9661.977,E2 -9661.977} C_VEL
LIN {X 0,Y 429.243,Z 335.293,A -85,B 0,C 180,E1 -9663.589,E2 -9663.589} C_VEL
LIN {X 0,Y 428.828,Z 348.645,A -85,B 0,C 180,E1 -9664.019,E2 -9664.019} C_VEL
LIN {X 0,Y 428.493,Z 360.845,A -85,B 0,C 180,E1 -9664.6,E2 -9664.6} C_VEL
LIN {X 0,Y 427.932,Z 372.867,A -85,B 0,C 180,E1 -9665.37,E2 -9665.37} C_VEL
LIN {X 0,Y 427.305,Z 384.171,A -85,B 0,C 180,E1 -9666.302,E2 -9666.302} C_VEL
LIN {X 0,Y 426.694,Z 394.764,A -85,B 0,C 180,E1 -9667.394,E2 -9667.394} C_VEL
LIN {X 0,Y 426.002,Z 404.7,A -85,B 0,C 180,E1 -9668.677,E2 -9668.677} C_VEL
LIN {X 0,Y 425.518,Z 413.534,A -85,B 0,C 180,E1 -9670.096,E2 -9670.096} C_VEL
LIN {X 0,Y 424.99,Z 421.211,A -85,B 0,C 180,E1 -9671.649,E2 -9671.649} C_VEL
LIN {X 0,Y 424.664,Z 427.435,A -85,B 0,C 180,E1 -9673.266,E2 -9673.266} C_VEL
LIN {X 0,Y 424.463,Z 431.426,A -85,B 0,C 180,E1 -9674.605,E2 -9674.605} C_VEL
LIN {X 0,Y 424.276,Z 434.428,A -85,B 0,C 180,E1 -9675.916,E2 -9675.916} C_VEL
LIN {X 0,Y 424.154,Z 436.579,A -85,B 0,C 180,E1 -9677.208,E2 -9677.208} C_VEL
LIN {X 0,Y 424.103,Z 437.92,A -85,B 0,C 180,E1 -9678.482,E2 -9678.482} C_VEL
LIN {X 0,Y 424.046,Z 438.52,A -85,B 0,C 180,E1 -9679.732,E2 -9679.732} C_VEL
LIN {X 0,Y 424.016,Z 438.37,A -85,B 0,C 180,E1 -9681.163,E2 -9681.163} C_VEL
LIN {X 0,Y 424.101,Z 437.195,A -85,B 0,C 180,E1 -9682.688,E2 -9682.688} C_VEL
LIN {X 0,Y 424.336,Z 434.29,A -85,B 0,C 180,E1 -9684.572,E2 -9684.572} C_VEL
LIN {X 0,Y 424.587,Z 429.824,A -85,B 0,C 180,E1 -9686.385,E2 -9686.385} C_VEL
LIN {X 0,Y 425.016,Z 424.15,A -85,B 0,C 180,E1 -9688.053,E2 -9688.053} C_VEL
LIN {X 0,Y 425.458,Z 417.842,A -85,B 0,C 180,E1 -9689.493,E2 -9689.493} C_VEL
LIN {X 0,Y 426.037,Z 409.791,A -85,B 0,C 180,E1 -9690.951,E2 -9690.951} C_VEL
LIN {X 0,Y 426.733,Z 400.721,A -85,B 0,C 180,E1 -9692.273,E2 -9692.273} C_VEL
LIN {X 0,Y 427.27,Z 391.525,A -85,B 0,C 180,E1 -9693.371,E2 -9693.371} C_VEL
LIN {X 0,Y 428.009,Z 380.639,A -85,B 0,C 180,E1 -9694.409,E2 -9694.409} C_VEL
LIN {X 0,Y 428.691,Z 368.991,A -85,B 0,C 180,E1 -9695.289,E2 -9695.289} C_VEL
LIN {X 0,Y 429.191,Z 358.197,A -85,B 0,C 180,E1 -9695.923,E2 -9695.923} C_VEL
LIN {X 0,Y 429.589,Z 345.358,A -85,B 0,C 180,E1 -9696.481,E2 -9696.481} C_VEL
LIN {X 0,Y 429.93,Z 332.224,A -85,B 0,C 180,E1 -9696.844,E2 -9696.844} C_VEL
LIN {X 0,Y 431.137,Z 245.702,A -85,B 0,C 180,E1 -9698.428,E2 -9698.428} C_VEL
LIN {X 0,Y 427.282,Z 228.02,A -85,B 0,C 180,E1 -9698.994,E2 -9698.994} C_VEL
LIN {X 0,Y 426.975,Z 224.209,A -85,B 0,C 180,E1 -9699.778,E2 -9699.778} C_VEL
LIN {X 0,Y 425.34,Z 216.506,A -85,B 0,C 180,E1 -9701.454,E2 -9701.454} C_VEL
LIN {X 0,Y 425.31,Z 216.509,A -85,B 0,C 180,E1 -9704.67,E2 -9704.67} C_VEL
LIN {X 0,Y 425.386,Z 216.503,A -85,B 0,C 180,E1 -9707.598,E2 -9707.598} C_VEL
LIN {X 0,Y 425.396,Z 216.499,A -85,B 0,C 180,E1 -9711.449,E2 -9711.449} C_VEL
LIN {X 0,Y 425.533,Z 216.477,A -85,B 0,C 180,E1 -9714.313,E2 -9714.313} C_VEL
LIN {X 0,Y 425.523,Z 216.478,A -85,B 0,C 180,E1 -9718.107,E2 -9718.107} C_VEL
LIN {X 0,Y 425.651,Z 216.463,A -85,B 0,C 180,E1 -9720,E2 -9720} C_VEL
LIN {X 0,Y 425.496,Z 216.485,A -85,B 0,C 180,E1 -9722.841,E2 -9722.841} C_VEL
LIN {X 0,Y 425.477,Z 216.484,A -85,B 0,C 180,E1 -9726.64,E2 -9726.64} C_VEL
LIN {X 0,Y 425.357,Z 216.499,A -85,B 0,C 180,E1 -9729.511,E2 -9729.511} C_VEL
LIN {X 0,Y 425.36,Z 216.502,A -85,B 0,C 180,E1 -9732.911,E2 -9732.911} C_VEL
LIN {X 0,Y 425.327,Z 216.505,A -85,B 0,C 180,E1 -9736.61,E2 -9736.61} C_VEL
LIN {X 0,Y 425.286,Z 216.506,A -85,B 0,C 180,E1 -9739.637,E2 -9739.637} C_VEL
LIN {X 0,Y 425.249,Z 216.515,A -85,B 0,C 180,E1 -9742.341,E2 -9742.341} C_VEL
LIN {X 0,Y 425.256,Z 216.51,A -85,B 0,C 180,E1 -9745.448,E2 -9745.448} C_VEL
LIN {X 0,Y 425.294,Z 216.508,A -85,B 0,C 180,E1 -9748.635,E2 -9748.635} C_VEL
LIN {X 0,Y 425.23,Z 216.515,A -85,B 0,C 180,E1 -9751.93,E2 -9751.93} C_VEL
LIN {X 0,Y 425.269,Z 216.505,A -85,B 0,C 180,E1 -9755.339,E2 -9755.339} C_VEL
LIN {X 0,Y 425.264,Z 216.511,A -85,B 0,C 180,E1 -9758.903,E2 -9758.903} C_VEL
LIN {X 0,Y 425.262,Z 216.513,A -85,B 0,C 180,E1 -9761.961,E2 -9761.961} C_VEL
LIN {X 0,Y 425.263,Z 216.508,A -85,B 0,C 180,E1 -9765.287,E2 -9765.287} C_VEL
LIN {X 0,Y 425.254,Z 216.513,A -85,B 0,C 180,E1 -9768.625,E2 -9768.625} C_VEL
LIN {X 0,Y 425.285,Z 216.508,A -85,B 0,C 180,E1 -9771.105,E2 -9771.105} C_VEL
LIN {X 0,Y 425.286,Z 216.508,A -85,B 0,C 180,E1 -9774.667,E2 -9774.667} C_VEL
LIN {X 0,Y 425.253,Z 216.515,A -85,B 0,C 180,E1 -9778.076,E2 -9778.076} C_VEL
LIN {X 0,Y 425.322,Z 216.508,A -85,B 0,C 180,E1 -9781.371,E2 -9781.371} C_VEL
LIN {X 0,Y 425.361,Z 216.551,A -85,B 0,C 180,E1 -9782.246,E2 -9782.246} C_VEL
LIN {X 0,Y 427.86,Z 228.757,A -85,B 0,C 180,E1 -9784.721,E2 -9784.721} C_VEL
LIN {X 0,Y 428.268,Z 232.924,A -85,B 0,C 180,E1 -9785.524,E2 -9785.524} C_VEL
LIN {X 0,Y 427.264,Z 249.518,A -85,B 0,C 180,E1 -9788.534,E2 -9788.534} C_VEL
LIN {X 0,Y 426.583,Z 263.432,A -85,B 0,C 180,E1 -9791.038,E2 -9791.038} C_VEL
LIN {X 0,Y 430.226,Z 286.799,A -85,B 0,C 180,E1 -9791.669,E2 -9791.669} C_VEL
LIN {X 0,Y 430.664,Z 291.582,A -85,B 0,C 180,E1 -9791.782,E2 -9791.782} C_VEL
LIN {X 0,Y 429.614,Z 372.957,A -85,B 0,C 180,E1 -9793.275,E2 -9793.275} C_VEL
LIN {X 0,Y 428.997,Z 386.635,A -85,B 0,C 180,E1 -9793.709,E2 -9793.709} C_VEL
LIN {X 0,Y 428.379,Z 399.07,A -85,B 0,C 180,E1 -9794.296,E2 -9794.296} C_VEL
LIN {X 0,Y 427.736,Z 410.239,A -85,B 0,C 180,E1 -9795.004,E2 -9795.004} C_VEL
LIN {X 0,Y 427.017,Z 421.642,A -85,B 0,C 180,E1 -9795.928,E2 -9795.928} C_VEL
LIN {X 0,Y 426.266,Z 432.428,A -85,B 0,C 180,E1 -9797.02,E2 -9797.02} C_VEL
LIN {X 0,Y 425.731,Z 441.059,A -85,B 0,C 180,E1 -9798.093,E2 -9798.093} C_VEL
LIN {X 0,Y 425.168,Z 449.031,A -85,B 0,C 180,E1 -9799.284,E2 -9799.284} C_VEL
LIN {X 0,Y 424.712,Z 456.827,A -85,B 0,C 180,E1 -9800.716,E2 -9800.716} C_VEL
LIN {X 0,Y 424.365,Z 464.036,A -85,B 0,C 180,E1 -9802.387,E2 -9802.387} C_VEL
LIN {X 0,Y 424.222,Z 468.559,A -85,B 0,C 180,E1 -9803.727,E2 -9803.727} C_VEL
LIN {X 0,Y 424.199,Z 472.513,A -85,B 0,C 180,E1 -9805.249,E2 -9805.249} C_VEL
LIN {X 0,Y 424.109,Z 474.391,A -85,B 0,C 180,E1 -9806.2,E2 -9806.2} C_VEL
LIN {X 0,Y 424.177,Z 475.812,A -85,B 0,C 180,E1 -9807.151,E2 -9807.151} C_VEL
LIN {X 0,Y 424.166,Z 476.826,A -85,B 0,C 180,E1 -9808.101,E2 -9808.101} C_VEL
LIN {X 0,Y 424.139,Z 477.442,A -85,B 0,C 180,E1 -9809.051,E2 -9809.051} C_VEL
LIN {X 0,Y 424.14,Z 477.628,A -85,B 0,C 180,E1 -9810,E2 -9810} C_VEL
LIN {X 0,Y 424.139,Z 477.388,A -85,B 0,C 180,E1 -9810.949,E2 -9810.949} C_VEL
LIN {X 0,Y 424.165,Z 476.754,A -85,B 0,C 180,E1 -9811.899,E2 -9811.899} C_VEL
LIN {X 0,Y 424.175,Z 475.719,A -85,B 0,C 180,E1 -9812.849,E2 -9812.849} C_VEL
LIN {X 0,Y 424.107,Z 474.225,A -85,B 0,C 180,E1 -9813.8,E2 -9813.8} C_VEL
LIN {X 0,Y 424.22,Z 471.173,A -85,B 0,C 180,E1 -9815.227,E2 -9815.227} C_VEL
LIN {X 0,Y 424.299,Z 467.031,A -85,B 0,C 180,E1 -9816.657,E2 -9816.657} C_VEL
LIN {X 0,Y 424.511,Z 460.669,A -85,B 0,C 180,E1 -9818.328,E2 -9818.328} C_VEL
LIN {X 0,Y 424.839,Z 453.731,A -85,B 0,C 180,E1 -9819.761,E2 -9819.761} C_VEL
LIN {X 0,Y 425.218,Z 446.64,A -85,B 0,C 180,E1 -9820.956,E2 -9820.956} C_VEL
LIN {X 0,Y 425.781,Z 438.096,A -85,B 0,C 180,E1 -9822.147,E2 -9822.147} C_VEL
LIN {X 0,Y 426.452,Z 427.527,A -85,B 0,C 180,E1 -9823.338,E2 -9823.338} C_VEL
LIN {X 0,Y 427.116,Z 415.631,A -85,B 0,C 180,E1 -9824.409,E2 -9824.409} C_VEL
LIN {X 0,Y 427.787,Z 403.667,A -85,B 0,C 180,E1 -9825.238,E2 -9825.238} C_VEL
LIN {X 0,Y 428.4,Z 391.272,A -85,B 0,C 180,E1 -9825.886,E2 -9825.886} C_VEL
LIN {X 0,Y 428.923,Z 378.594,A -85,B 0,C 180,E1 -9826.355,E2 -9826.355} C_VEL
LIN {X 0,Y 429.271,Z 363.832,A -85,B 0,C 180,E1 -9826.678,E2 -9826.678} C_VEL
LIN {X 0,Y 429.994,Z 289.565,A -85,B 0,C 180,E1 -9828.003,E2 -9828.003} C_VEL
LIN {X 0,Y 426.42,Z 264.941,A -85,B 0,C 180,E1 -9828.619,E2 -9828.619} C_VEL
LIN {X 0,Y 427.468,Z 246.89,A -85,B 0,C 180,E1 -9831.962,E2 -9831.962} C_VEL
LIN {X 0,Y 428.326,Z 232.122,A -85,B 0,C 180,E1 -9834.731,E2 -9834.731} C_VEL
LIN {X 0,Y 427.161,Z 225.295,A -85,B 0,C 180,E1 -9836.108,E2 -9836.108} C_VEL
LIN {X 0,Y 425.386,Z 216.5,A -85,B 0,C 180,E1 -9837.953,E2 -9837.953} C_VEL
LIN {X 0,Y 425.277,Z 216.51,A -85,B 0,C 180,E1 -9840.813,E2 -9840.813} C_VEL
LIN {X 0,Y 425.298,Z 216.508,A -85,B 0,C 180,E1 -9844.285,E2 -9844.285} C_VEL
LIN {X 0,Y 425.262,Z 216.513,A -85,B 0,C 180,E1 -9847.691,E2 -9847.691} C_VEL
LIN {X 0,Y 425.26,Z 216.51,A -85,B 0,C 180,E1 -9850.517,E2 -9850.517} C_VEL
LIN {X 0,Y 425.236,Z 216.514,A -85,B 0,C 180,E1 -9853.347,E2 -9853.347} C_VEL
LIN {X 0,Y 425.233,Z 216.512,A -85,B 0,C 180,E1 -9856.646,E2 -9856.646} C_VEL
LIN {X 0,Y 425.258,Z 216.514,A -85,B 0,C 180,E1 -9859.869,E2 -9859.869} C_VEL
LIN {X 0,Y 425.247,Z 216.51,A -85,B 0,C 180,E1 -9862.486,E2 -9862.486} C_VEL
LIN {X 0,Y 425.275,Z 216.511,A -85,B 0,C 180,E1 -9865.814,E2 -9865.814} C_VEL
LIN {X 0,Y 425.255,Z 216.513,A -85,B 0,C 180,E1 -9869.236,E2 -9869.236} C_VEL
LIN {X 0,Y 425.311,Z 216.502,A -85,B 0,C 180,E1 -9872.439,E2 -9872.439} C_VEL
LIN {X 0,Y 425.311,Z 216.507,A -85,B 0,C 180,E1 -9875.599,E2 -9875.599} C_VEL
LIN {X 0,Y 425.25,Z 216.511,A -85,B 0,C 180,E1 -9878.679,E2 -9878.679} C_VEL
LIN {X 0,Y 425.288,Z 216.508,A -85,B 0,C 180,E1 -9881.7,E2 -9881.7} C_VEL
LIN {X 0,Y 425.3,Z 216.505,A -85,B 0,C 180,E1 -9884.669,E2 -9884.669} C_VEL
LIN {X 0,Y 425.383,Z 216.496,A -85,B 0,C 180,E1 -9887.597,E2 -9887.597} C_VEL
LIN {X 0,Y 425.395,Z 216.495,A -85,B 0,C 180,E1 -9891.449,E2 -9891.449} C_VEL
LIN {X 0,Y 425.498,Z 216.479,A -85,B 0,C 180,E1 -9894.312,E2 -9894.312} C_VEL
LIN {X 0,Y 425.522,Z 216.476,A -85,B 0,C 180,E1 -9898.107,E2 -9898.107} C_VEL
LIN {X 0,Y 425.65,Z 216.46,A -85,B 0,C 180,E1 -9900,E2 -9900} C_VEL
LIN {X 0,Y 425.497,Z 216.486,A -85,B 0,C 180,E1 -9902.84,E2 -9902.84} C_VEL
LIN {X 0,Y 425.534,Z 216.475,A -85,B 0,C 180,E1 -9905.687,E2 -9905.687} C_VEL
LIN {X 0,Y 425.395,Z 216.496,A -85,B 0,C 180,E1 -9908.551,E2 -9908.551} C_VEL
LIN {X 0,Y 425.385,Z 216.497,A -85,B 0,C 180,E1 -9912.402,E2 -9912.402} C_VEL
LIN {X 0,Y 425.352,Z 216.501,A -85,B 0,C 180,E1 -9916.313,E2 -9916.313} C_VEL
LIN {X 0,Y 425.332,Z 216.5,A -85,B 0,C 180,E1 -9919.655,E2 -9919.655} C_VEL
LIN {X 0,Y 425.325,Z 216.506,A -85,B 0,C 180,E1 -9922.336,E2 -9922.336} C_VEL
LIN {X 0,Y 425.26,Z 216.509,A -85,B 0,C 180,E1 -9925.447,E2 -9925.447} C_VEL
LIN {X 0,Y 425.299,Z 216.508,A -85,B 0,C 180,E1 -9928.634,E2 -9928.634} C_VEL
LIN {X 0,Y 425.228,Z 216.515,A -85,B 0,C 180,E1 -9931.93,E2 -9931.93} C_VEL
LIN {X 0,Y 425.265,Z 216.508,A -85,B 0,C 180,E1 -9935.339,E2 -9935.339} C_VEL
LIN {X 0,Y 425.283,Z 216.506,A -85,B 0,C 180,E1 -9939.049,E2 -9939.049} C_VEL
LIN {X 0,Y 425.302,Z 216.505,A -85,B 0,C 180,E1 -9942.649,E2 -9942.649} C_VEL
LIN {X 0,Y 425.237,Z 216.519,A -85,B 0,C 180,E1 -9946.047,E2 -9946.047} C_VEL
LIN {X 0,Y 425.28,Z 216.507,A -85,B 0,C 180,E1 -9948.628,E2 -9948.628} C_VEL
LIN {X 0,Y 425.3,Z 216.504,A -85,B 0,C 180,E1 -9951.107,E2 -9951.107} C_VEL
LIN {X 0,Y 425.282,Z 216.506,A -85,B 0,C 180,E1 -9954.667,E2 -9954.667} C_VEL
LIN {X 0,Y 425.251,Z 216.514,A -85,B 0,C 180,E1 -9958.076,E2 -9958.076} C_VEL
LIN {X 0,Y 425.325,Z 216.503,A -85,B 0,C 180,E1 -9961.371,E2 -9961.371} C_VEL
LIN {X 0,Y 425.285,Z 216.506,A -85,B 0,C 180,E1 -9964.557,E2 -9964.557} C_VEL
LIN {X 0,Y 425.279,Z 216.513,A -85,B 0,C 180,E1 -9967.664,E2 -9967.664} C_VEL
LIN {X 0,Y 425.355,Z 216.497,A -85,B 0,C 180,E1 -9970.706,E2 -9970.706} C_VEL
LIN {X 0,Y 425.383,Z 216.499,A -85,B 0,C 180,E1 -9973.69,E2 -9973.69} C_VEL
LIN {X 0,Y 425.408,Z 216.496,A -85,B 0,C 180,E1 -9977.6,E2 -9977.6} C_VEL
LIN {X 0,Y 425.44,Z 216.493,A -85,B 0,C 180,E1 -9981.451,E2 -9981.451} C_VEL
LIN {X 0,Y 425.548,Z 216.473,A -85,B 0,C 180,E1 -9984.314,E2 -9984.314} C_VEL
LIN {X 0,Y 425.573,Z 216.47,A -85,B 0,C 180,E1 -9988.108,E2 -9988.108} C_VEL
LIN {X 0,Y 425.7,Z 216.454,A -85,B 0,C 180,E1 -9990,E2 -9990} C_VEL
LIN {X 0,Y 425.555,Z 216.475,A -85,B 0,C 180,E1 -9992.84,E2 -9992.84} C_VEL
LIN {X 0,Y 425.543,Z 216.475,A -85,B 0,C 180,E1 -9995.686,E2 -9995.686} C_VEL
LIN {X 0,Y 425.434,Z 216.489,A -85,B 0,C 180,E1 -9998.549,E2 -9998.549} C_VEL
LIN {X 0,Y 425.397,Z 216.492,A -85,B 0,C 180,E1 -9999.196,E2 -9999.196} C_VEL
LIN {X 0,Y 424.73,Z 216.578,A -85,B 0,C 180,E1 -9999.986,E2 -9999.986} C_VEL
LIN {X 0,Y 421.88,Z 216.938,A -85,B 0,C 180,E1 -10001.27,E2 -10001.27} C_VEL
LIN {X 0,Y 419.46,Z 217.24,A -85,B 0,C 180,E1 -10002.306,E2 -10002.306} C_VEL
LIN {X 0,Y 418.408,Z 217.368,A -85,B 0,C 180,E1 -10003.106,E2 -10003.106} C_VEL
LIN {X 0,Y 418.316,Z 217.376,A -85,B 0,C 180,E1 -10003.378,E2 -10003.378} C_VEL
LIN {X 0,Y 418.308,Z 217.38,A -85,B 0,C 180,E1 -10006.734,E2 -10006.734} C_VEL
LIN {X 0,Y 418.264,Z 217.38,A -85,B 0,C 180,E1 -10009.788,E2 -10009.788} C_VEL
LIN {X 0,Y 418.224,Z 217.392,A -85,B 0,C 180,E1 -10012.734,E2 -10012.734} C_VEL
LIN {X 0,Y 418.26,Z 217.384,A -85,B 0,C 180,E1 -10015.902,E2 -10015.902} C_VEL
LIN {X 0,Y 418.365,Z 217.578,A -85,B 0,C 180,E1 -10018.738,E2 -10018.738} C_VEL
LIN {X 0,Y 419.854,Z 225.741,A -85,B 0,C 180,E1 -10020.696,E2 -10020.696} C_VEL
LIN {X 0,Y 419.881,Z 227.874,A -85,B 0,C 180,E1 -10021.183,E2 -10021.183} C_VEL
LIN {X 0,Y 423.634,Z 246.651,A -85,B 0,C 180,E1 -10021.719,E2 -10021.719} C_VEL
LIN {X 0,Y 422.373,Z 335.945,A -85,B 0,C 180,E1 -10023.361,E2 -10023.361} C_VEL
LIN {X 0,Y 421.93,Z 349.593,A -85,B 0,C 180,E1 -10023.814,E2 -10023.814} C_VEL
LIN {X 0,Y 421.591,Z 361.446,A -85,B 0,C 180,E1 -10024.395,E2 -10024.395} C_VEL
LIN {X 0,Y 420.996,Z 373.715,A -85,B 0,C 180,E1 -10025.202,E2 -10025.202} C_VEL
LIN {X 0,Y 420.294,Z 385.821,A -85,B 0,C 180,E1 -10026.232,E2 -10026.232} C_VEL
LIN {X 0,Y 419.626,Z 396.404,A -85,B 0,C 180,E1 -10027.377,E2 -10027.377} C_VEL
LIN {X 0,Y 418.965,Z 405.722,A -85,B 0,C 180,E1 -10028.624,E2 -10028.624} C_VEL
LIN {X 0,Y 418.522,Z 413.705,A -85,B 0,C 180,E1 -10029.935,E2 -10029.935} C_VEL
LIN {X 0,Y 418.023,Z 420.393,A -85,B 0,C 180,E1 -10031.276,E2 -10031.276} C_VEL
LIN {X 0,Y 417.648,Z 426.978,A -85,B 0,C 180,E1 -10032.951,E2 -10032.951} C_VEL
LIN {X 0,Y 417.416,Z 431.161,A -85,B 0,C 180,E1 -10034.316,E2 -10034.316} C_VEL
LIN {X 0,Y 417.234,Z 434.353,A -85,B 0,C 180,E1 -10035.663,E2 -10035.663} C_VEL
LIN {X 0,Y 417.124,Z 435.757,A -85,B 0,C 180,E1 -10036.42,E2 -10036.42} C_VEL
LIN {X 0,Y 417.02,Z 437.7,A -85,B 0,C 180,E1 -10037.855,E2 -10037.855} C_VEL
LIN {X 0,Y 416.949,Z 438.744,A -85,B 0,C 180,E1 -10039.326,E2 -10039.326} C_VEL
LIN {X 0,Y 416.943,Z 438.843,A -85,B 0,C 180,E1 -10040.832,E2 -10040.832} C_VEL
LIN {X 0,Y 417.012,Z 437.655,A -85,B 0,C 180,E1 -10042.648,E2 -10042.648} C_VEL
LIN {X 0,Y 417.249,Z 434.925,A -85,B 0,C 180,E1 -10044.51,E2 -10044.51} C_VEL
LIN {X 0,Y 417.483,Z 430.927,A -85,B 0,C 180,E1 -10046.253,E2 -10046.253} C_VEL
LIN {X 0,Y 417.947,Z 425.21,A -85,B 0,C 180,E1 -10048.016,E2 -10048.016} C_VEL
LIN {X 0,Y 418.338,Z 419.648,A -85,B 0,C 180,E1 -10049.357,E2 -10049.357} C_VEL
LIN {X 0,Y 419.003,Z 411.695,A -85,B 0,C 180,E1 -10050.895,E2 -10050.895} C_VEL
LIN {X 0,Y 419.733,Z 402.335,A -85,B 0,C 180,E1 -10052.324,E2 -10052.324} C_VEL
LIN {X 0,Y 420.369,Z 392.249,A -85,B 0,C 180,E1 -10053.568,E2 -10053.568} C_VEL
LIN {X 0,Y 421.106,Z 382.352,A -85,B 0,C 180,E1 -10054.549,E2 -10054.549} C_VEL
LIN {X 0,Y 421.841,Z 370.271,A -85,B 0,C 180,E1 -10055.497,E2 -10055.497} C_VEL
LIN {X 0,Y 422.414,Z 358.65,A -85,B 0,C 180,E1 -10056.202,E2 -10056.202} C_VEL
LIN {X 0,Y 422.854,Z 345.477,A -85,B 0,C 180,E1 -10056.783,E2 -10056.783} C_VEL
LIN {X 0,Y 423.244,Z 331.766,A -85,B 0,C 180,E1 -10057.161,E2 -10057.161} C_VEL
LIN {X 0,Y 424.564,Z 246.983,A -85,B 0,C 180,E1 -10058.739,E2 -10058.739} C_VEL
LIN {X 0,Y 420.442,Z 228.352,A -85,B 0,C 180,E1 -10059.357,E2 -10059.357} C_VEL
LIN {X 0,Y 418.888,Z 220.068,A -85,B 0,C 180,E1 -10061.158,E2 -10061.158} C_VEL
LIN {X 0,Y 418.271,Z 217.386,A -85,B 0,C 180,E1 -10061.763,E2 -10061.763} C_VEL
LIN {X 0,Y 418.266,Z 217.386,A -85,B 0,C 180,E1 -10064.405,E2 -10064.405} C_VEL
LIN {X 0,Y 418.326,Z 217.384,A -85,B 0,C 180,E1 -10067.385,E2 -10067.385} C_VEL
LIN {X 0,Y 418.299,Z 217.381,A -85,B 0,C 180,E1 -10070.328,E2 -10070.328} C_VEL
LIN {X 0,Y 418.453,Z 217.363,A -85,B 0,C 180,E1 -10073.249,E2 -10073.249} C_VEL
LIN {X 0,Y 418.297,Z 217.382,A -85,B 0,C 180,E1 -10075.181,E2 -10075.181} C_VEL
LIN {X 0,Y 418.493,Z 217.354,A -85,B 0,C 180,E1 -10078.076,E2 -10078.076} C_VEL
LIN {X 0,Y 418.621,Z 217.338,A -85,B 0,C 180,E1 -10080,E2 -10080} C_VEL
LIN {X 0,Y 418.451,Z 217.362,A -85,B 0,C 180,E1 -10082.888,E2 -10082.888} C_VEL
LIN {X 0,Y 418.441,Z 217.362,A -85,B 0,C 180,E1 -10086.752,E2 -10086.752} C_VEL
LIN {X 0,Y 418.298,Z 217.378,A -85,B 0,C 180,E1 -10089.673,E2 -10089.673} C_VEL
LIN {X 0,Y 418.311,Z 217.379,A -85,B 0,C 180,E1 -10093.007,E2 -10093.007} C_VEL
LIN {X 0,Y 418.277,Z 217.382,A -85,B 0,C 180,E1 -10096.74,E2 -10096.74} C_VEL
LIN {X 0,Y 418.229,Z 217.385,A -85,B 0,C 180,E1 -10099.791,E2 -10099.791} C_VEL
LIN {X 0,Y 418.193,Z 217.392,A -85,B 0,C 180,E1 -10102.739,E2 -10102.739} C_VEL
LIN {X 0,Y 418.233,Z 217.386,A -85,B 0,C 180,E1 -10105.907,E2 -10105.907} C_VEL
LIN {X 0,Y 418.23,Z 217.383,A -85,B 0,C 180,E1 -10109.165,E2 -10109.165} C_VEL
LIN {X 0,Y 418.225,Z 217.388,A -85,B 0,C 180,E1 -10112.847,E2 -10112.847} C_VEL
LIN {X 0,Y 418.215,Z 217.39,A -85,B 0,C 180,E1 -10116.241,E2 -10116.241} C_VEL
LIN {X 0,Y 418.216,Z 217.389,A -85,B 0,C 180,E1 -10119.686,E2 -10119.686} C_VEL
LIN {X 0,Y 418.202,Z 217.392,A -85,B 0,C 180,E1 -10122.324,E2 -10122.324} C_VEL
LIN {X 0,Y 418.214,Z 217.386,A -85,B 0,C 180,E1 -10125.112,E2 -10125.112} C_VEL
LIN {X 0,Y 418.219,Z 217.388,A -85,B 0,C 180,E1 -10127.77,E2 -10127.77} C_VEL
LIN {X 0,Y 418.232,Z 217.388,A -85,B 0,C 180,E1 -10130.623,E2 -10130.623} C_VEL
LIN {X 0,Y 418.229,Z 217.391,A -85,B 0,C 180,E1 -10133.979,E2 -10133.979} C_VEL
LIN {X 0,Y 418.246,Z 217.386,A -85,B 0,C 180,E1 -10137.159,E2 -10137.159} C_VEL
LIN {X 0,Y 418.26,Z 217.388,A -85,B 0,C 180,E1 -10140.898,E2 -10140.898} C_VEL
LIN {X 0,Y 418.324,Z 217.473,A -85,B 0,C 180,E1 -10141.942,E2 -10141.942} C_VEL
LIN {X 0,Y 420.812,Z 229.311,A -85,B 0,C 180,E1 -10144.404,E2 -10144.404} C_VEL
LIN {X 0,Y 421.397,Z 234.152,A -85,B 0,C 180,E1 -10145.361,E2 -10145.361} C_VEL
LIN {X 0,Y 420.334,Z 250.725,A -85,B 0,C 180,E1 -10148.42,E2 -10148.42} C_VEL
LIN {X 0,Y 419.679,Z 263.031,A -85,B 0,C 180,E1 -10150.673,E2 -10150.673} C_VEL
LIN {X 0,Y 423.272,Z 285.433,A -85,B 0,C 180,E1 -10151.3,E2 -10151.3} C_VEL
LIN {X 0,Y 423.979,Z 293.065,A -85,B 0,C 180,E1 -10151.484,E2 -10151.484} C_VEL
LIN {X 0,Y 422.847,Z 373.365,A -85,B 0,C 180,E1 -10152.999,E2 -10152.999} C_VEL
LIN {X 0,Y 422.197,Z 386.753,A -85,B 0,C 180,E1 -10153.439,E2 -10153.439} C_VEL
LIN {X 0,Y 421.568,Z 399.041,A -85,B 0,C 180,E1 -10154.035,E2 -10154.035} C_VEL
LIN {X 0,Y 420.766,Z 411.716,A -85,B 0,C 180,E1 -10154.873,E2 -10154.873} C_VEL
LIN {X 0,Y 420.015,Z 423.039,A -85,B 0,C 180,E1 -10155.835,E2 -10155.835} C_VEL
LIN {X 0,Y 419.241,Z 433.287,A -85,B 0,C 180,E1 -10156.922,E2 -10156.922} C_VEL
LIN {X 0,Y 418.625,Z 442.538,A -85,B 0,C 180,E1 -10158.133,E2 -10158.133} C_VEL
LIN {X 0,Y 417.95,Z 451.576,A -85,B 0,C 180,E1 -10159.587,E2 -10159.587} C_VEL
LIN {X 0,Y 417.526,Z 458.85,A -85,B 0,C 180,E1 -10161.044,E2 -10161.044} C_VEL
LIN {X 0,Y 417.258,Z 465.489,A -85,B 0,C 180,E1 -10162.743,E2 -10162.743} C_VEL
LIN {X 0,Y 417.085,Z 469.884,A -85,B 0,C 180,E1 -10164.198,E2 -10164.198} C_VEL
LIN {X 0,Y 417.105,Z 472.223,A -85,B 0,C 180,E1 -10165.168,E2 -10165.168} C_VEL
LIN {X 0,Y 417.024,Z 474.087,A -85,B 0,C 180,E1 -10166.135,E2 -10166.135} C_VEL
LIN {X 0,Y 417.073,Z 475.502,A -85,B 0,C 180,E1 -10167.103,E2 -10167.103} C_VEL
LIN {X 0,Y 417.091,Z 476.513,A -85,B 0,C 180,E1 -10168.069,E2 -10168.069} C_VEL
LIN {X 0,Y 417.058,Z 477.123,A -85,B 0,C 180,E1 -10169.034,E2 -10169.034} C_VEL
LIN {X 0,Y 417.057,Z 477.295,A -85,B 0,C 180,E1 -10170,E2 -10170} C_VEL
LIN {X 0,Y 417.058,Z 477.05,A -85,B 0,C 180,E1 -10170.965,E2 -10170.965} C_VEL
LIN {X 0,Y 417.091,Z 476.408,A -85,B 0,C 180,E1 -10171.931,E2 -10171.931} C_VEL
LIN {X 0,Y 417.073,Z 475.363,A -85,B 0,C 180,E1 -10172.897,E2 -10172.897} C_VEL
LIN {X 0,Y 417.022,Z 473.853,A -85,B 0,C 180,E1 -10173.865,E2 -10173.865} C_VEL
LIN {X 0,Y 417.131,Z 470.781,A -85,B 0,C 180,E1 -10175.316,E2 -10175.316} C_VEL
LIN {X 0,Y 417.231,Z 466.618,A -85,B 0,C 180,E1 -10176.771,E2 -10176.771} C_VEL
LIN {X 0,Y 417.453,Z 460.228,A -85,B 0,C 180,E1 -10178.47,E2 -10178.47} C_VEL
LIN {X 0,Y 417.795,Z 453.26,A -85,B 0,C 180,E1 -10179.927,E2 -10179.927} C_VEL
LIN {X 0,Y 418.219,Z 446.133,A -85,B 0,C 180,E1 -10181.141,E2 -10181.141} C_VEL
LIN {X 0,Y 418.775,Z 437.526,A -85,B 0,C 180,E1 -10182.354,E2 -10182.354} C_VEL
LIN {X 0,Y 419.503,Z 426.891,A -85,B 0,C 180,E1 -10183.563,E2 -10183.563} C_VEL
LIN {X 0,Y 420.106,Z 416.356,A -85,B 0,C 180,E1 -10184.531,E2 -10184.531} C_VEL
LIN {X 0,Y 420.795,Z 404.778,A -85,B 0,C 180,E1 -10185.373,E2 -10185.373} C_VEL
LIN {X 0,Y 421.495,Z 391.521,A -85,B 0,C 180,E1 -10186.092,E2 -10186.092} C_VEL
